LIN {X 0,Y 446.51,Z 528.86,A -85,B 0,C 180,E1 -8628.193,E2 -8628.193} C_VEL
LIN {X 0,Y 446.592,Z 528.855,A -85,B 0,C 180,E1 -8631.858,E2 -8631.858} C_VEL
LIN {X 0,Y 446.639,Z 528.845,A -85,B 0,C 180,E1 -8634.582,E2 -8634.582} C_VEL
LIN {X 0,Y 446.702,Z 528.834,A -85,B 0,C 180,E1 -8637.295,E2 -8637.295} C_VEL
LIN {X 0,Y 446.787,Z 528.83,A -85,B 0,C 180,E1 -8640,E2 -8640} C_VEL
LIN {X 0,Y 446.703,Z 528.834,A -85,B 0,C 180,E1 -8642.705,E2 -8642.705} C_VEL
LIN {X 0,Y 446.639,Z 528.846,A -85,B 0,C 180,E1 -8646.324,E2 -8646.324} C_VEL
LIN {X 0,Y 446.531,Z 528.859,A -85,B 0,C 180,E1 -8649.055,E2 -8649.055} C_VEL
LIN {X 0,Y 446.526,Z 528.859,A -85,B 0,C 180,E1 -8652.73,E2 -8652.73} C_VEL
LIN {X 0,Y 446.482,Z 528.86,A -85,B 0,C 180,E1 -8656.459,E2 -8656.459} C_VEL
LIN {X 0,Y 446.462,Z 528.872,A -85,B 0,C 180,E1 -8659.304,E2 -8659.304} C_VEL
LIN {X 0,Y 446.411,Z 528.873,A -85,B 0,C 180,E1 -8662.2,E2 -8662.2} C_VEL
LIN {X 0,Y 446.452,Z 528.872,A -85,B 0,C 180,E1 -8665.153,E2 -8665.153} C_VEL
LIN {X 0,Y 446.478,Z 528.868,A -85,B 0,C 180,E1 -8668.179,E2 -8668.179} C_VEL
LIN {X 0,Y 446.428,Z 528.877,A -85,B 0,C 180,E1 -8671.779,E2 -8671.779} C_VEL
LIN {X 0,Y 446.425,Z 528.871,A -85,B 0,C 180,E1 -8675.054,E2 -8675.054} C_VEL
LIN {X 0,Y 446.425,Z 528.874,A -85,B 0,C 180,E1 -8678.083,E2 -8678.083} C_VEL
LIN {X 0,Y 446.422,Z 528.873,A -85,B 0,C 180,E1 -8680.918,E2 -8680.918} C_VEL
LIN {X 0,Y 446.412,Z 528.878,A -85,B 0,C 180,E1 -8683.845,E2 -8683.845} C_VEL
LIN {X 0,Y 446.442,Z 528.867,A -85,B 0,C 180,E1 -8686.398,E2 -8686.398} C_VEL
LIN {X 0,Y 446.465,Z 528.87,A -85,B 0,C 180,E1 -8689.806,E2 -8689.806} C_VEL
LIN {X 0,Y 446.429,Z 528.859,A -85,B 0,C 180,E1 -8692.125,E2 -8692.125} C_VEL
LIN {X 0,Y 446.428,Z 528.877,A -85,B 0,C 180,E1 -8695.478,E2 -8695.478} C_VEL
LIN {X 0,Y 446.414,Z 528.831,A -85,B 0,C 180,E1 -8698.701,E2 -8698.701} C_VEL
LIN {X 0,Y 446.483,Z 528.871,A -85,B 0,C 180,E1 -8701.822,E2 -8701.822} C_VEL
LIN {X 0,Y 446.527,Z 529.058,A -85,B 0,C 180,E1 -8703.557,E2 -8703.557} C_VEL
LIN {X 0,Y 448.792,Z 540.632,A -85,B 0,C 180,E1 -8705.975,E2 -8705.975} C_VEL
LIN {X 0,Y 449.081,Z 544.438,A -85,B 0,C 180,E1 -8706.725,E2 -8706.725} C_VEL
LIN {X 0,Y 448.095,Z 560.858,A -85,B 0,C 180,E1 -8709.816,E2 -8709.816} C_VEL
LIN {X 0,Y 447.517,Z 573.5,A -85,B 0,C 180,E1 -8712.138,E2 -8712.138} C_VEL
LIN {X 0,Y 450.897,Z 595.443,A -85,B 0,C 180,E1 -8712.662,E2 -8712.662} C_VEL
LIN {X 0,Y 450.108,Z 681.533,A -85,B 0,C 180,E1 -8714.056,E2 -8714.056} C_VEL
LIN {X 0,Y 449.652,Z 694.781,A -85,B 0,C 180,E1 -8714.447,E2 -8714.447} C_VEL
LIN {X 0,Y 449.113,Z 708.062,A -85,B 0,C 180,E1 -8715.037,E2 -8715.037} C_VEL
LIN {X 0,Y 448.566,Z 719.218,A -85,B 0,C 180,E1 -8715.715,E2 -8715.715} C_VEL
LIN {X 0,Y 447.922,Z 730.654,A -85,B 0,C 180,E1 -8716.605,E2 -8716.605} C_VEL
LIN {X 0,Y 447.407,Z 741.258,A -85,B 0,C 180,E1 -8717.643,E2 -8717.643} C_VEL
LIN {X 0,Y 446.849,Z 749.797,A -85,B 0,C 180,E1 -8718.663,E2 -8718.663} C_VEL
LIN {X 0,Y 446.393,Z 757.677,A -85,B 0,C 180,E1 -8719.799,E2 -8719.799} C_VEL
LIN {X 0,Y 445.992,Z 765.376,A -85,B 0,C 180,E1 -8721.163,E2 -8721.163} C_VEL
LIN {X 0,Y 445.668,Z 772.472,A -85,B 0,C 180,E1 -8722.753,E2 -8722.753} C_VEL
LIN {X 0,Y 445.494,Z 776.598,A -85,B 0,C 180,E1 -8723.926,E2 -8723.926} C_VEL
LIN {X 0,Y 445.417,Z 780.807,A -85,B 0,C 180,E1 -8725.476,E2 -8725.476} C_VEL
LIN {X 0,Y 445.381,Z 782.669,A -85,B 0,C 180,E1 -8726.382,E2 -8726.382} C_VEL
LIN {X 0,Y 445.433,Z 784.067,A -85,B 0,C 180,E1 -8727.288,E2 -8727.288} C_VEL
LIN {X 0,Y 445.338,Z 785.666,A -85,B 0,C 180,E1 -8729.097,E2 -8729.097} C_VEL
LIN {X 0,Y 445.342,Z 785.882,A -85,B 0,C 180,E1 -8730.001,E2 -8730.001} C_VEL
LIN {X 0,Y 445.338,Z 785.664,A -85,B 0,C 180,E1 -8730.905,E2 -8730.905} C_VEL
LIN {X 0,Y 445.433,Z 784.061,A -85,B 0,C 180,E1 -8732.714,E2 -8732.714} C_VEL
LIN {X 0,Y 445.381,Z 782.661,A -85,B 0,C 180,E1 -8733.62,E2 -8733.62} C_VEL
LIN {X 0,Y 445.482,Z 779.728,A -85,B 0,C 180,E1 -8734.978,E2 -8734.978} C_VEL
LIN {X 0,Y 445.576,Z 774.321,A -85,B 0,C 180,E1 -8736.749,E2 -8736.749} C_VEL
LIN {X 0,Y 445.848,Z 768.627,A -85,B 0,C 180,E1 -8738.157,E2 -8738.157} C_VEL
LIN {X 0,Y 446.16,Z 761.723,A -85,B 0,C 180,E1 -8739.521,E2 -8739.521} C_VEL
LIN {X 0,Y 446.611,Z 753.086,A -85,B 0,C 180,E1 -8740.886,E2 -8740.886} C_VEL
LIN {X 0,Y 447.213,Z 744.234,A -85,B 0,C 180,E1 -8742.019,E2 -8742.019} C_VEL
LIN {X 0,Y 447.682,Z 735.241,A -85,B 0,C 180,E1 -8742.972,E2 -8742.972} C_VEL
LIN {X 0,Y 448.293,Z 723.88,A -85,B 0,C 180,E1 -8743.948,E2 -8743.948} C_VEL
LIN {X 0,Y 448.894,Z 712.012,A -85,B 0,C 180,E1 -8744.74,E2 -8744.74} C_VEL
LIN {X 0,Y 449.493,Z 699.667,A -85,B 0,C 180,E1 -8745.357,E2 -8745.357} C_VEL
LIN {X 0,Y 449.947,Z 686.981,A -85,B 0,C 180,E1 -8745.806,E2 -8745.806} C_VEL
LIN {X 0,Y 450.202,Z 673.707,A -85,B 0,C 180,E1 -8746.087,E2 -8746.087} C_VEL
LIN {X 0,Y 450.721,Z 593.516,A -85,B 0,C 180,E1 -8747.374,E2 -8747.374} C_VEL
LIN {X 0,Y 447.503,Z 573.499,A -85,B 0,C 180,E1 -8747.859,E2 -8747.859} C_VEL
LIN {X 0,Y 448.186,Z 559.56,A -85,B 0,C 180,E1 -8750.421,E2 -8750.421} C_VEL
LIN {X 0,Y 449.08,Z 544.406,A -85,B 0,C 180,E1 -8753.276,E2 -8753.276} C_VEL
LIN {X 0,Y 448.611,Z 539.586,A -85,B 0,C 180,E1 -8754.233,E2 -8754.233} C_VEL
LIN {X 0,Y 446.536,Z 529.053,A -85,B 0,C 180,E1 -8756.444,E2 -8756.444} C_VEL
LIN {X 0,Y 446.452,Z 528.857,A -85,B 0,C 180,E1 -8759.21,E2 -8759.21} C_VEL
LIN {X 0,Y 446.426,Z 528.879,A -85,B 0,C 180,E1 -8762.362,E2 -8762.362} C_VEL
LIN {X 0,Y 446.423,Z 528.875,A -85,B 0,C 180,E1 -8765.626,E2 -8765.626} C_VEL
LIN {X 0,Y 446.448,Z 528.872,A -85,B 0,C 180,E1 -8769.027,E2 -8769.027} C_VEL
LIN {X 0,Y 446.438,Z 528.875,A -85,B 0,C 180,E1 -8772.278,E2 -8772.278} C_VEL
LIN {X 0,Y 446.455,Z 528.872,A -85,B 0,C 180,E1 -8775.104,E2 -8775.104} C_VEL
LIN {X 0,Y 446.431,Z 528.876,A -85,B 0,C 180,E1 -8778.609,E2 -8778.609} C_VEL
LIN {X 0,Y 446.464,Z 528.87,A -85,B 0,C 180,E1 -8780.975,E2 -8780.975} C_VEL
LIN {X 0,Y 446.424,Z 528.88,A -85,B 0,C 180,E1 -8784.374,E2 -8784.374} C_VEL
LIN {X 0,Y 446.426,Z 528.877,A -85,B 0,C 180,E1 -8787.639,E2 -8787.639} C_VEL
LIN {X 0,Y 446.453,Z 528.876,A -85,B 0,C 180,E1 -8790.791,E2 -8790.791} C_VEL
LIN {X 0,Y 446.536,Z 529.061,A -85,B 0,C 180,E1 -8792.271,E2 -8792.271} C_VEL
LIN {X 0,Y 448.78,Z 539.14,A -85,B 0,C 180,E1 -8793.993,E2 -8793.993} C_VEL
LIN {X 0,Y 449.498,Z 544.011,A -85,B 0,C 180,E1 -8794.782,E2 -8794.782} C_VEL
LIN {X 0,Y 448.867,Z 564.635,A -85,B 0,C 180,E1 -8797.928,E2 -8797.928} C_VEL
LIN {X 0,Y 448.11,Z 586.321,A -85,B 0,C 180,E1 -8801.245,E2 -8801.245} C_VEL
LIN {X 0,Y 447.44,Z 609.001,A -85,B 0,C 180,E1 -8804.746,E2 -8804.746} C_VEL
LIN {X 0,Y 447.231,Z 616.994,A -85,B 0,C 180,E1 -8805.934,E2 -8805.934} C_VEL
LIN {X 0,Y 448.935,Z 631.407,A -85,B 0,C 180,E1 -8806.294,E2 -8806.294} C_VEL
LIN {X 0,Y 448.157,Z 697.089,A -85,B 0,C 180,E1 -8807.548,E2 -8807.548} C_VEL
LIN {X 0,Y 447.884,Z 707.461,A -85,B 0,C 180,E1 -8807.885,E2 -8807.885} C_VEL
LIN {X 0,Y 447.61,Z 717.158,A -85,B 0,C 180,E1 -8808.337,E2 -8808.337} C_VEL
LIN {X 0,Y 447.278,Z 728.032,A -85,B 0,C 180,E1 -8809.017,E2 -8809.017} C_VEL
LIN {X 0,Y 446.889,Z 737.516,A -85,B 0,C 180,E1 -8809.809,E2 -8809.809} C_VEL
LIN {X 0,Y 446.624,Z 744.205,A -85,B 0,C 180,E1 -8810.49,E2 -8810.49} C_VEL
LIN {X 0,Y 446.26,Z 751.577,A -85,B 0,C 180,E1 -8811.396,E2 -8811.396} C_VEL
LIN {X 0,Y 445.99,Z 757.653,A -85,B 0,C 180,E1 -8812.302,E2 -8812.302} C_VEL
LIN {X 0,Y 445.825,Z 763.632,A -85,B 0,C 180,E1 -8813.393,E2 -8813.393} C_VEL
LIN {X 0,Y 445.656,Z 768.771,A -85,B 0,C 180,E1 -8814.571,E2 -8814.571} C_VEL
LIN {X 0,Y 445.485,Z 773.124,A -85,B 0,C 180,E1 -8815.929,E2 -8815.929} C_VEL
LIN {X 0,Y 445.449,Z 776.133,A -85,B 0,C 180,E1 -8817.287,E2 -8817.287} C_VEL
LIN {X 0,Y 445.356,Z 777.465,A -85,B 0,C 180,E1 -8818.191,E2 -8818.191} C_VEL
LIN {X 0,Y 445.314,Z 778.286,A -85,B 0,C 180,E1 -8819.096,E2 -8819.096} C_VEL
LIN {X 0,Y 445.315,Z 778.581,A -85,B 0,C 180,E1 -8820,E2 -8820} C_VEL
LIN {X 0,Y 445.315,Z 778.281,A -85,B 0,C 180,E1 -8820.904,E2 -8820.904} C_VEL
LIN {X 0,Y 445.357,Z 777.461,A -85,B 0,C 180,E1 -8821.809,E2 -8821.809} C_VEL
LIN {X 0,Y 445.449,Z 776.132,A -85,B 0,C 180,E1 -8822.713,E2 -8822.713} C_VEL
LIN {X 0,Y 445.465,Z 773.118,A -85,B 0,C 180,E1 -8824.071,E2 -8824.071} C_VEL
LIN {X 0,Y 445.625,Z 768.766,A -85,B 0,C 180,E1 -8825.43,E2 -8825.43} C_VEL
LIN {X 0,Y 445.781,Z 763.037,A -85,B 0,C 180,E1 -8826.725,E2 -8826.725} C_VEL
LIN {X 0,Y 445.94,Z 757.662,A -85,B 0,C 180,E1 -8827.699,E2 -8827.699} C_VEL
LIN {X 0,Y 446.211,Z 751.59,A -85,B 0,C 180,E1 -8828.605,E2 -8828.605} C_VEL
LIN {X 0,Y 446.515,Z 744.23,A -85,B 0,C 180,E1 -8829.513,E2 -8829.513} C_VEL
LIN {X 0,Y 446.924,Z 735.167,A -85,B 0,C 180,E1 -8830.419,E2 -8830.419} C_VEL
LIN {X 0,Y 447.32,Z 724.744,A -85,B 0,C 180,E1 -8831.211,E2 -8831.211} C_VEL
LIN {X 0,Y 447.566,Z 716.17,A -85,B 0,C 180,E1 -8831.722,E2 -8831.722} C_VEL
LIN {X 0,Y 447.778,Z 706.821,A -85,B 0,C 180,E1 -8832.147,E2 -8832.147} C_VEL
LIN {X 0,Y 448.033,Z 696.114,A -85,B 0,C 180,E1 -8832.485,E2 -8832.485} C_VEL
LIN {X 0,Y 448.615,Z 629.959,A -85,B 0,C 180,E1 -8833.69,E2 -8833.69} C_VEL
LIN {X 0,Y 447.022,Z 616.645,A -85,B 0,C 180,E1 -8834.006,E2 -8834.006} C_VEL
LIN {X 0,Y 447.552,Z 598.063,A -85,B 0,C 180,E1 -8836.901,E2 -8836.901} C_VEL
LIN {X 0,Y 448.343,Z 577.229,A -85,B 0,C 180,E1 -8840.173,E2 -8840.173} C_VEL
LIN {X 0,Y 449.038,Z 557.569,A -85,B 0,C 180,E1 -8843.278,E2 -8843.278} C_VEL
LIN {X 0,Y 449.527,Z 545.318,A -85,B 0,C 180,E1 -8845.216,E2 -8845.216} C_VEL
LIN {X 0,Y 448.529,Z 538.743,A -85,B 0,C 180,E1 -8846.316,E2 -8846.316} C_VEL
LIN {X 0,Y 446.533,Z 528.964,A -85,B 0,C 180,E1 -8848.027,E2 -8848.027} C_VEL
LIN {X 0,Y 446.42,Z 528.879,A -85,B 0,C 180,E1 -8851.3,E2 -8851.3} C_VEL
LIN {X 0,Y 446.433,Z 528.873,A -85,B 0,C 180,E1 -8854.523,E2 -8854.523} C_VEL
LIN {X 0,Y 446.434,Z 528.872,A -85,B 0,C 180,E1 -8858.082,E2 -8858.082} C_VEL
LIN {X 0,Y 446.427,Z 528.861,A -85,B 0,C 180,E1 -8860.917,E2 -8860.917} C_VEL
LIN {X 0,Y 446.403,Z 528.866,A -85,B 0,C 180,E1 -8863.846,E2 -8863.846} C_VEL
LIN {X 0,Y 446.402,Z 528.876,A -85,B 0,C 180,E1 -8866.403,E2 -8866.403} C_VEL
LIN {X 0,Y 446.431,Z 528.864,A -85,B 0,C 180,E1 -8869.082,E2 -8869.082} C_VEL
LIN {X 0,Y 446.411,Z 528.872,A -85,B 0,C 180,E1 -8872.121,E2 -8872.121} C_VEL
LIN {X 0,Y 446.427,Z 528.871,A -85,B 0,C 180,E1 -8875.476,E2 -8875.476} C_VEL
LIN {X 0,Y 446.42,Z 528.875,A -85,B 0,C 180,E1 -8878.699,E2 -8878.699} C_VEL
LIN {X 0,Y 446.489,Z 528.867,A -85,B 0,C 180,E1 -8881.821,E2 -8881.821} C_VEL
LIN {X 0,Y 446.454,Z 528.871,A -85,B 0,C 180,E1 -8884.847,E2 -8884.847} C_VEL
LIN {X 0,Y 446.478,Z 529.008,A -85,B 0,C 180,E1 -8887.437,E2 -8887.437} C_VEL
LIN {X 0,Y 448.136,Z 537.779,A -85,B 0,C 180,E1 -8889.577,E2 -8889.577} C_VEL
LIN {X 0,Y 448.116,Z 539.979,A -85,B 0,C 180,E1 -8890.073,E2 -8890.073} C_VEL
LIN {X 0,Y 447.429,Z 543.234,A -85,B 0,C 180,E1 -8890.675,E2 -8890.675} C_VEL
LIN {X 0,Y 445.584,Z 548.544,A -85,B 0,C 180,E1 -8891.354,E2 -8891.354} C_VEL
LIN {X 0,Y 443.803,Z 554.744,A -85,B 0,C 180,E1 -8891.883,E2 -8891.883} C_VEL
LIN {X 0,Y 443.187,Z 559.936,A -85,B 0,C 180,E1 -8892.167,E2 -8892.167} C_VEL
LIN {X 0,Y 443.431,Z 563.572,A -85,B 0,C 180,E1 -8892.287,E2 -8892.287} C_VEL
LIN {X 0,Y 444.253,Z 568.245,A -85,B 0,C 180,E1 -8892.399,E2 -8892.399} C_VEL
LIN {X 0,Y 443.384,Z 657.163,A -85,B 0,C 180,E1 -8893.865,E2 -8893.865} C_VEL
LIN {X 0,Y 442.99,Z 671.026,A -85,B 0,C 180,E1 -8894.294,E2 -8894.294} C_VEL
LIN {X 0,Y 442.503,Z 683.424,A -85,B 0,C 180,E1 -8894.866,E2 -8894.866} C_VEL
LIN {X 0,Y 441.942,Z 695.269,A -85,B 0,C 180,E1 -8895.612,E2 -8895.612} C_VEL
LIN {X 0,Y 441.388,Z 706.671,A -85,B 0,C 180,E1 -8896.537,E2 -8896.537} C_VEL
LIN {X 0,Y 440.768,Z 716.867,A -85,B 0,C 180,E1 -8897.569,E2 -8897.569} C_VEL
LIN {X 0,Y 440.149,Z 726.052,A -85,B 0,C 180,E1 -8898.72,E2 -8898.72} C_VEL
LIN {X 0,Y 439.552,Z 734.97,A -85,B 0,C 180,E1 -8900.102,E2 -8900.102} C_VEL
LIN {X 0,Y 439.104,Z 742.146,A -85,B 0,C 180,E1 -8901.485,E2 -8901.485} C_VEL
LIN {X 0,Y 438.788,Z 746.99,A -85,B 0,C 180,E1 -8902.637,E2 -8902.637} C_VEL
LIN {X 0,Y 438.686,Z 751.69,A -85,B 0,C 180,E1 -8904.022,E2 -8904.022} C_VEL
LIN {X 0,Y 438.424,Z 755.291,A -85,B 0,C 180,E1 -8905.402,E2 -8905.402} C_VEL
LIN {X 0,Y 438.428,Z 757.148,A -85,B 0,C 180,E1 -8906.323,E2 -8906.323} C_VEL
LIN {X 0,Y 438.395,Z 758.551,A -85,B 0,C 180,E1 -8907.243,E2 -8907.243} C_VEL
LIN {X 0,Y 438.255,Z 760.167,A -85,B 0,C 180,E1 -8909.08,E2 -8909.08} C_VEL
LIN {X 0,Y 438.254,Z 760.402,A -85,B 0,C 180,E1 -8909.999,E2 -8909.999} C_VEL
LIN {X 0,Y 438.255,Z 760.216,A -85,B 0,C 180,E1 -8910.918,E2 -8910.918} C_VEL
LIN {X 0,Y 438.392,Z 758.667,A -85,B 0,C 180,E1 -8912.756,E2 -8912.756} C_VEL
LIN {X 0,Y 438.413,Z 757.314,A -85,B 0,C 180,E1 -8913.676,E2 -8913.676} C_VEL
LIN {X 0,Y 438.481,Z 754.45,A -85,B 0,C 180,E1 -8915.057,E2 -8915.057} C_VEL
LIN {X 0,Y 438.693,Z 750.563,A -85,B 0,C 180,E1 -8916.438,E2 -8916.438} C_VEL
LIN {X 0,Y 438.902,Z 745.555,A -85,B 0,C 180,E1 -8917.822,E2 -8917.822} C_VEL
LIN {X 0,Y 439.321,Z 739.248,A -85,B 0,C 180,E1 -8919.205,E2 -8919.205} C_VEL
LIN {X 0,Y 439.803,Z 731.349,A -85,B 0,C 180,E1 -8920.588,E2 -8920.588} C_VEL
LIN {X 0,Y 440.285,Z 723.299,A -85,B 0,C 180,E1 -8921.742,E2 -8921.742} C_VEL
LIN {X 0,Y 441.015,Z 713.467,A -85,B 0,C 180,E1 -8922.89,E2 -8922.89} C_VEL
LIN {X 0,Y 441.542,Z 702.694,A -85,B 0,C 180,E1 -8923.907,E2 -8923.907} C_VEL
LIN {X 0,Y 442.135,Z 691.584,A -85,B 0,C 180,E1 -8924.733,E2 -8924.733} C_VEL
LIN {X 0,Y 442.709,Z 679.604,A -85,B 0,C 180,E1 -8925.42,E2 -8925.42} C_VEL
LIN {X 0,Y 443.122,Z 666.471,A -85,B 0,C 180,E1 -8925.966,E2 -8925.966} C_VEL
LIN {X 0,Y 443.533,Z 653.261,A -85,B 0,C 180,E1 -8926.305,E2 -8926.305} C_VEL
LIN {X 0,Y 444.113,Z 567.022,A -85,B 0,C 180,E1 -8927.721,E2 -8927.721} C_VEL
LIN {X 0,Y 440.768,Z 550.156,A -85,B 0,C 180,E1 -8928.171,E2 -8928.171} C_VEL
LIN {X 0,Y 440.78,Z 547.921,A -85,B 0,C 180,E1 -8928.595,E2 -8928.595} C_VEL
LIN {X 0,Y 441.2,Z 539.437,A -85,B 0,C 180,E1 -8930.513,E2 -8930.513} C_VEL
LIN {X 0,Y 439.437,Z 529.822,A -85,B 0,C 180,E1 -8932.912,E2 -8932.912} C_VEL
LIN {X 0,Y 439.433,Z 529.742,A -85,B 0,C 180,E1 -8936.41,E2 -8936.41} C_VEL
LIN {X 0,Y 439.417,Z 529.744,A -85,B 0,C 180,E1 -8938.672,E2 -8938.672} C_VEL
LIN {X 0,Y 439.369,Z 529.753,A -85,B 0,C 180,E1 -8942.03,E2 -8942.03} C_VEL
LIN {X 0,Y 439.394,Z 529.752,A -85,B 0,C 180,E1 -8945.34,E2 -8945.34} C_VEL
LIN {X 0,Y 439.387,Z 529.75,A -85,B 0,C 180,E1 -8948.593,E2 -8948.593} C_VEL
LIN {X 0,Y 439.386,Z 529.751,A -85,B 0,C 180,E1 -8951.256,E2 -8951.256} C_VEL
LIN {X 0,Y 439.401,Z 529.741,A -85,B 0,C 180,E1 -8954.728,E2 -8954.728} C_VEL
LIN {X 0,Y 439.393,Z 529.752,A -85,B 0,C 180,E1 -8957.795,E2 -8957.795} C_VEL
LIN {X 0,Y 439.447,Z 529.734,A -85,B 0,C 180,E1 -8960.229,E2 -8960.229} C_VEL
LIN {X 0,Y 439.373,Z 529.756,A -85,B 0,C 180,E1 -8963.712,E2 -8963.712} C_VEL
LIN {X 0,Y 439.367,Z 529.754,A -85,B 0,C 180,E1 -8967.053,E2 -8967.053} C_VEL
LIN {X 0,Y 439.39,Z 529.749,A -85,B 0,C 180,E1 -8970.275,E2 -8970.275} C_VEL
LIN {X 0,Y 439.427,Z 529.748,A -85,B 0,C 180,E1 -8973.588,E2 -8973.588} C_VEL
LIN {X 0,Y 439.38,Z 529.748,A -85,B 0,C 180,E1 -8976.429,E2 -8976.429} C_VEL
LIN {X 0,Y 439.382,Z 529.752,A -85,B 0,C 180,E1 -8979.397,E2 -8979.397} C_VEL
LIN {X 0,Y 439.424,Z 529.741,A -85,B 0,C 180,E1 -8982.309,E2 -8982.309} C_VEL
LIN {X 0,Y 439.44,Z 529.741,A -85,B 0,C 180,E1 -8985.174,E2 -8985.174} C_VEL
LIN {X 0,Y 439.476,Z 529.738,A -85,B 0,C 180,E1 -8988.001,E2 -8988.001} C_VEL
LIN {X 0,Y 439.54,Z 529.734,A -85,B 0,C 180,E1 -8991.726,E2 -8991.726} C_VEL
LIN {X 0,Y 439.614,Z 529.72,A -85,B 0,C 180,E1 -8994.496,E2 -8994.496} C_VEL
LIN {X 0,Y 439.628,Z 529.718,A -85,B 0,C 180,E1 -8998.168,E2 -8998.168} C_VEL
LIN {X 0,Y 439.757,Z 529.706,A -85,B 0,C 180,E1 -9000,E2 -9000} C_VEL
LIN {X 0,Y 439.649,Z 529.712,A -85,B 0,C 180,E1 -9002.749,E2 -9002.749} C_VEL
LIN {X 0,Y 439.61,Z 529.721,A -85,B 0,C 180,E1 -9006.425,E2 -9006.425} C_VEL
LIN {X 0,Y 439.493,Z 529.737,A -85,B 0,C 180,E1 -9009.202,E2 -9009.202} C_VEL
LIN {X 0,Y 439.496,Z 529.735,A -85,B 0,C 180,E1 -9012.727,E2 -9012.727} C_VEL
LIN {X 0,Y 439.44,Z 529.737,A -85,B 0,C 180,E1 -9016.349,E2 -9016.349} C_VEL
LIN {X 0,Y 439.424,Z 529.751,A -85,B 0,C 180,E1 -9019.625,E2 -9019.625} C_VEL
LIN {X 0,Y 439.358,Z 529.75,A -85,B 0,C 180,E1 -9022.576,E2 -9022.576} C_VEL
LIN {X 0,Y 439.399,Z 529.752,A -85,B 0,C 180,E1 -9025.585,E2 -9025.585} C_VEL
LIN {X 0,Y 439.411,Z 529.747,A -85,B 0,C 180,E1 -9028.674,E2 -9028.674} C_VEL
LIN {X 0,Y 439.375,Z 529.754,A -85,B 0,C 180,E1 -9032.034,E2 -9032.034} C_VEL
LIN {X 0,Y 439.39,Z 529.748,A -85,B 0,C 180,E1 -9035.342,E2 -9035.342} C_VEL
LIN {X 0,Y 439.385,Z 529.749,A -85,B 0,C 180,E1 -9038.595,E2 -9038.595} C_VEL
LIN {X 0,Y 439.383,Z 529.752,A -85,B 0,C 180,E1 -9041.258,E2 -9041.258} C_VEL
LIN {X 0,Y 439.4,Z 529.748,A -85,B 0,C 180,E1 -9044.73,E2 -9044.73} C_VEL
LIN {X 0,Y 439.409,Z 529.749,A -85,B 0,C 180,E1 -9047.799,E2 -9047.799} C_VEL
LIN {X 0,Y 439.447,Z 529.739,A -85,B 0,C 180,E1 -9050.231,E2 -9050.231} C_VEL
LIN {X 0,Y 439.374,Z 529.748,A -85,B 0,C 180,E1 -9053.714,E2 -9053.714} C_VEL
LIN {X 0,Y 439.37,Z 529.733,A -85,B 0,C 180,E1 -9057.055,E2 -9057.055} C_VEL
LIN {X 0,Y 439.38,Z 529.723,A -85,B 0,C 180,E1 -9060.275,E2 -9060.275} C_VEL
LIN {X 0,Y 439.47,Z 529.836,A -85,B 0,C 180,E1 -9063.272,E2 -9063.272} C_VEL
LIN {X 0,Y 441.813,Z 541.718,A -85,B 0,C 180,E1 -9065.821,E2 -9065.821} C_VEL
LIN {X 0,Y 442.142,Z 545.523,A -85,B 0,C 180,E1 -9066.586,E2 -9066.586} C_VEL
LIN {X 0,Y 441.101,Z 562.606,A -85,B 0,C 180,E1 -9069.856,E2 -9069.856} C_VEL
LIN {X 0,Y 440.59,Z 573.219,A -85,B 0,C 180,E1 -9071.841,E2 -9071.841} C_VEL
LIN {X 0,Y 442.189,Z 582.977,A -85,B 0,C 180,E1 -9072.105,E2 -9072.105} C_VEL
LIN {X 0,Y 444.109,Z 596.39,A -85,B 0,C 180,E1 -9072.407,E2 -9072.407} C_VEL
LIN {X 0,Y 443.298,Z 681.339,A -85,B 0,C 180,E1 -9073.805,E2 -9073.805} C_VEL
LIN {X 0,Y 442.821,Z 694.584,A -85,B 0,C 180,E1 -9074.201,E2 -9074.201} C_VEL
LIN {X 0,Y 442.312,Z 706.741,A -85,B 0,C 180,E1 -9074.743,E2 -9074.743} C_VEL
LIN {X 0,Y 441.681,Z 719.017,A -85,B 0,C 180,E1 -9075.487,E2 -9075.487} C_VEL
LIN {X 0,Y 441.048,Z 729.687,A -85,B 0,C 180,E1 -9076.323,E2 -9076.323} C_VEL
LIN {X 0,Y 440.443,Z 741.055,A -85,B 0,C 180,E1 -9077.444,E2 -9077.444} C_VEL
LIN {X 0,Y 439.873,Z 749.594,A -85,B 0,C 180,E1 -9078.48,E2 -9078.48} C_VEL
LIN {X 0,Y 439.371,Z 757.473,A -85,B 0,C 180,E1 -9079.634,E2 -9079.634} C_VEL
LIN {X 0,Y 438.937,Z 765.171,A -85,B 0,C 180,E1 -9081.02,E2 -9081.02} C_VEL
LIN {X 0,Y 438.606,Z 772.267,A -85,B 0,C 180,E1 -9082.636,E2 -9082.636} C_VEL
LIN {X 0,Y 438.393,Z 776.825,A -85,B 0,C 180,E1 -9083.967,E2 -9083.967} C_VEL
LIN {X 0,Y 438.346,Z 780.603,A -85,B 0,C 180,E1 -9085.403,E2 -9085.403} C_VEL
LIN {X 0,Y 438.283,Z 782.465,A -85,B 0,C 180,E1 -9086.323,E2 -9086.323} C_VEL
LIN {X 0,Y 438.341,Z 783.862,A -85,B 0,C 180,E1 -9087.244,E2 -9087.244} C_VEL
LIN {X 0,Y 438.252,Z 785.462,A -85,B 0,C 180,E1 -9089.082,E2 -9089.082} C_VEL
LIN {X 0,Y 438.253,Z 785.678,A -85,B 0,C 180,E1 -9090.001,E2 -9090.001} C_VEL
LIN {X 0,Y 438.278,Z 784.851,A -85,B 0,C 180,E1 -9091.839,E2 -9091.839} C_VEL
LIN {X 0,Y 438.341,Z 783.856,A -85,B 0,C 180,E1 -9092.758,E2 -9092.758} C_VEL
LIN {X 0,Y 438.283,Z 782.456,A -85,B 0,C 180,E1 -9093.678,E2 -9093.678} C_VEL
LIN {X 0,Y 438.392,Z 779.522,A -85,B 0,C 180,E1 -9095.059,E2 -9095.059} C_VEL
LIN {X 0,Y 438.449,Z 775.547,A -85,B 0,C 180,E1 -9096.443,E2 -9096.443} C_VEL
LIN {X 0,Y 438.724,Z 769.433,A -85,B 0,C 180,E1 -9098.058,E2 -9098.058} C_VEL
LIN {X 0,Y 439.066,Z 762.753,A -85,B 0,C 180,E1 -9099.444,E2 -9099.444} C_VEL
LIN {X 0,Y 439.523,Z 754.467,A -85,B 0,C 180,E1 -9100.83,E2 -9100.83} C_VEL
LIN {X 0,Y 440.111,Z 745.977,A -85,B 0,C 180,E1 -9101.982,E2 -9101.982} C_VEL
LIN {X 0,Y 440.68,Z 735.869,A -85,B 0,C 180,E1 -9103.098,E2 -9103.098} C_VEL
LIN {X 0,Y 441.295,Z 725.101,A -85,B 0,C 180,E1 -9104.057,E2 -9104.057} C_VEL
LIN {X 0,Y 441.922,Z 713.728,A -85,B 0,C 180,E1 -9104.86,E2 -9104.86} C_VEL
LIN {X 0,Y 442.536,Z 702.061,A -85,B 0,C 180,E1 -9105.487,E2 -9105.487} C_VEL
LIN {X 0,Y 443.031,Z 688.601,A -85,B 0,C 180,E1 -9106,E2 -9106} C_VEL
LIN {X 0,Y 443.398,Z 675.272,A -85,B 0,C 180,E1 -9106.311,E2 -9106.311} C_VEL
LIN {X 0,Y 443.994,Z 594.706,A -85,B 0,C 180,E1 -9107.622,E2 -9107.622} C_VEL
LIN {X 0,Y 440.562,Z 573.531,A -85,B 0,C 180,E1 -9108.133,E2 -9108.133} C_VEL
LIN {X 0,Y 440.689,Z 570.679,A -85,B 0,C 180,E1 -9108.6,E2 -9108.6} C_VEL
LIN {X 0,Y 441.86,Z 550.549,A -85,B 0,C 180,E1 -9112.442,E2 -9112.442} C_VEL
LIN {X 0,Y 442.137,Z 544.223,A -85,B 0,C 180,E1 -9113.664,E2 -9113.664} C_VEL
LIN {X 0,Y 440.358,Z 534.063,A -85,B 0,C 180,E1 -9115.776,E2 -9115.776} C_VEL
LIN {X 0,Y 439.482,Z 529.843,A -85,B 0,C 180,E1 -9116.729,E2 -9116.729} C_VEL
LIN {X 0,Y 439.386,Z 529.741,A -85,B 0,C 180,E1 -9119.726,E2 -9119.726} C_VEL
LIN {X 0,Y 439.376,Z 529.753,A -85,B 0,C 180,E1 -9122.946,E2 -9122.946} C_VEL
LIN {X 0,Y 439.377,Z 529.756,A -85,B 0,C 180,E1 -9126.287,E2 -9126.287} C_VEL
LIN {X 0,Y 439.405,Z 529.752,A -85,B 0,C 180,E1 -9129.849,E2 -9129.849} C_VEL
LIN {X 0,Y 439.385,Z 529.754,A -85,B 0,C 180,E1 -9132.627,E2 -9132.627} C_VEL
LIN {X 0,Y 439.403,Z 529.75,A -85,B 0,C 180,E1 -9135.271,E2 -9135.271} C_VEL
LIN {X 0,Y 439.392,Z 529.752,A -85,B 0,C 180,E1 -9138.743,E2 -9138.743} C_VEL
LIN {X 0,Y 439.389,Z 529.753,A -85,B 0,C 180,E1 -9141.606,E2 -9141.606} C_VEL
LIN {X 0,Y 439.404,Z 529.751,A -85,B 0,C 180,E1 -9144.844,E2 -9144.844} C_VEL
LIN {X 0,Y 439.376,Z 529.757,A -85,B 0,C 180,E1 -9148.14,E2 -9148.14} C_VEL
LIN {X 0,Y 439.458,Z 529.785,A -85,B 0,C 180,E1 -9151.792,E2 -9151.792} C_VEL
LIN {X 0,Y 439.61,Z 530.432,A -85,B 0,C 180,E1 -9152.024,E2 -9152.024} C_VEL
LIN {X 0,Y 441.68,Z 539.177,A -85,B 0,C 180,E1 -9153.542,E2 -9153.542} C_VEL
LIN {X 0,Y 442.705,Z 545.655,A -85,B 0,C 180,E1 -9154.619,E2 -9154.619} C_VEL
LIN {X 0,Y 442.015,Z 566.31,A -85,B 0,C 180,E1 -9157.813,E2 -9157.813} C_VEL
LIN {X 0,Y 441.186,Z 588.036,A -85,B 0,C 180,E1 -9161.181,E2 -9161.181} C_VEL
LIN {X 0,Y 440.478,Z 610.836,A -85,B 0,C 180,E1 -9164.736,E2 -9164.736} C_VEL
LIN {X 0,Y 440.288,Z 616.892,A -85,B 0,C 180,E1 -9165.646,E2 -9165.646} C_VEL
LIN {X 0,Y 442.102,Z 631.443,A -85,B 0,C 180,E1 -9166.043,E2 -9166.043} C_VEL
LIN {X 0,Y 441.214,Z 697.846,A -85,B 0,C 180,E1 -9167.348,E2 -9167.348} C_VEL
LIN {X 0,Y 440.964,Z 707.987,A -85,B 0,C 180,E1 -9167.692,E2 -9167.692} C_VEL
LIN {X 0,Y 440.668,Z 718.644,A -85,B 0,C 180,E1 -9168.209,E2 -9168.209} C_VEL
LIN {X 0,Y 440.208,Z 729.73,A -85,B 0,C 180,E1 -9168.955,E2 -9168.955} C_VEL
LIN {X 0,Y 439.913,Z 737.717,A -85,B 0,C 180,E1 -9169.646,E2 -9169.646} C_VEL
LIN {X 0,Y 439.625,Z 744.369,A -85,B 0,C 180,E1 -9170.337,E2 -9170.337} C_VEL
LIN {X 0,Y 439.236,Z 751.71,A -85,B 0,C 180,E1 -9171.257,E2 -9171.257} C_VEL
LIN {X 0,Y 438.94,Z 757.766,A -85,B 0,C 180,E1 -9172.178,E2 -9172.178} C_VEL
LIN {X 0,Y 438.769,Z 763.612,A -85,B 0,C 180,E1 -9173.262,E2 -9173.262} C_VEL
LIN {X 0,Y 438.602,Z 768.872,A -85,B 0,C 180,E1 -9174.483,E2 -9174.483} C_VEL
LIN {X 0,Y 438.389,Z 773.216,A -85,B 0,C 180,E1 -9175.863,E2 -9175.863} C_VEL
LIN {X 0,Y 438.379,Z 776.224,A -85,B 0,C 180,E1 -9177.243,E2 -9177.243} C_VEL
LIN {X 0,Y 438.279,Z 777.542,A -85,B 0,C 180,E1 -9178.162,E2 -9178.162} C_VEL
LIN {X 0,Y 438.229,Z 778.351,A -85,B 0,C 180,E1 -9179.081,E2 -9179.081} C_VEL
LIN {X 0,Y 438.227,Z 778.636,A -85,B 0,C 180,E1 -9180,E2 -9180} C_VEL
LIN {X 0,Y 438.23,Z 778.326,A -85,B 0,C 180,E1 -9180.919,E2 -9180.919} C_VEL
LIN {X 0,Y 438.28,Z 777.483,A -85,B 0,C 180,E1 -9181.838,E2 -9181.838} C_VEL
LIN {X 0,Y 438.361,Z 776.13,A -85,B 0,C 180,E1 -9182.757,E2 -9182.757} C_VEL
LIN {X 0,Y 438.372,Z 773.078,A -85,B 0,C 180,E1 -9184.137,E2 -9184.137} C_VEL
LIN {X 0,Y 438.551,Z 768.665,A -85,B 0,C 180,E1 -9185.518,E2 -9185.518} C_VEL
LIN {X 0,Y 438.707,Z 763.306,A -85,B 0,C 180,E1 -9186.749,E2 -9186.749} C_VEL
LIN {X 0,Y 438.894,Z 757.451,A -85,B 0,C 180,E1 -9187.823,E2 -9187.823} C_VEL
LIN {X 0,Y 439.16,Z 751.316,A -85,B 0,C 180,E1 -9188.745,E2 -9188.745} C_VEL
LIN {X 0,Y 439.555,Z 742.888,A -85,B 0,C 180,E1 -9189.781,E2 -9189.781} C_VEL
LIN {X 0,Y 439.993,Z 733.272,A -85,B 0,C 180,E1 -9190.701,E2 -9190.701} C_VEL
LIN {X 0,Y 440.315,Z 724.079,A -85,B 0,C 180,E1 -9191.392,E2 -9191.392} C_VEL
LIN {X 0,Y 440.611,Z 714.238,A -85,B 0,C 180,E1 -9191.968,E2 -9191.968} C_VEL
LIN {X 0,Y 440.87,Z 702.638,A -85,B 0,C 180,E1 -9192.457,E2 -9192.457} C_VEL
LIN {X 0,Y 441.142,Z 689.902,A -85,B 0,C 180,E1 -9192.771,E2 -9192.771} C_VEL
LIN {X 0,Y 441.605,Z 630.077,A -85,B 0,C 180,E1 -9193.88,E2 -9193.88} C_VEL
LIN {X 0,Y 440.009,Z 616.661,A -85,B 0,C 180,E1 -9194.207,E2 -9194.207} C_VEL
LIN {X 0,Y 440.583,Z 598.143,A -85,B 0,C 180,E1 -9197.116,E2 -9197.116} C_VEL
LIN {X 0,Y 441.402,Z 576.791,A -85,B 0,C 180,E1 -9200.505,E2 -9200.505} C_VEL
LIN {X 0,Y 442.143,Z 556.985,A -85,B 0,C 180,E1 -9203.663,E2 -9203.663} C_VEL
LIN {X 0,Y 442.576,Z 546.183,A -85,B 0,C 180,E1 -9205.389,E2 -9205.389} C_VEL
LIN {X 0,Y 440.813,Z 536.225,A -85,B 0,C 180,E1 -9207.085,E2 -9207.085} C_VEL
LIN {X 0,Y 439.484,Z 529.839,A -85,B 0,C 180,E1 -9208.236,E2 -9208.236} C_VEL
LIN {X 0,Y 439.377,Z 529.757,A -85,B 0,C 180,E1 -9211.86,E2 -9211.86} C_VEL
LIN {X 0,Y 439.404,Z 529.751,A -85,B 0,C 180,E1 -9215.156,E2 -9215.156} C_VEL
LIN {X 0,Y 439.392,Z 529.748,A -85,B 0,C 180,E1 -9218.594,E2 -9218.594} C_VEL
LIN {X 0,Y 439.386,Z 529.73,A -85,B 0,C 180,E1 -9221.256,E2 -9221.256} C_VEL
LIN {X 0,Y 439.403,Z 529.741,A -85,B 0,C 180,E1 -9224.729,E2 -9224.729} C_VEL
LIN {X 0,Y 439.4,Z 529.746,A -85,B 0,C 180,E1 -9227.795,E2 -9227.795} C_VEL
LIN {X 0,Y 439.393,Z 529.728,A -85,B 0,C 180,E1 -9230.223,E2 -9230.223} C_VEL
LIN {X 0,Y 439.377,Z 529.753,A -85,B 0,C 180,E1 -9233.712,E2 -9233.712} C_VEL
LIN {X 0,Y 439.376,Z 529.757,A -85,B 0,C 180,E1 -9237.054,E2 -9237.054} C_VEL
LIN {X 0,Y 439.387,Z 529.753,A -85,B 0,C 180,E1 -9240.274,E2 -9240.274} C_VEL
LIN {X 0,Y 439.433,Z 529.747,A -85,B 0,C 180,E1 -9243.396,E2 -9243.396} C_VEL
LIN {X 0,Y 439.424,Z 529.751,A -85,B 0,C 180,E1 -9246.93,E2 -9246.93} C_VEL
LIN {X 0,Y 439.445,Z 529.943,A -85,B 0,C 180,E1 -9247.242,E2 -9247.242} C_VEL
LIN {X 0,Y 441.174,Z 539.02,A -85,B 0,C 180,E1 -9249.484,E2 -9249.484} C_VEL
LIN {X 0,Y 440.75,Z 549.905,A -85,B 0,C 180,E1 -9251.899,E2 -9251.899} C_VEL
LIN {X 0,Y 441.535,Z 554.077,A -85,B 0,C 180,E1 -9252.048,E2 -9252.048} C_VEL
LIN {X 0,Y 443.431,Z 563.572,A -85,B 0,C 180,E1 -9252.287,E2 -9252.287} C_VEL
LIN {X 0,Y 443.24,Z 567.471,A -85,B 0,C 180,E1 -9252.344,E2 -9252.344} C_VEL
LIN {X 0,Y 440.801,Z 573.725,A -85,B 0,C 180,E1 -9252.347,E2 -9252.347} C_VEL
LIN {X 0,Y 438.037,Z 580.006,A -85,B 0,C 180,E1 -9252.336,E2 -9252.336} C_VEL
LIN {X 0,Y 437.382,Z 583.982,A -85,B 0,C 180,E1 -9252.376,E2 -9252.376} C_VEL
LIN {X 0,Y 436.576,Z 657.385,A -85,B 0,C 180,E1 -9253.607,E2 -9253.607} C_VEL
LIN {X 0,Y 436.184,Z 671.242,A -85,B 0,C 180,E1 -9254.042,E2 -9254.042} C_VEL
LIN {X 0,Y 435.667,Z 683.636,A -85,B 0,C 180,E1 -9254.623,E2 -9254.623} C_VEL
LIN {X 0,Y 435.064,Z 695.48,A -85,B 0,C 180,E1 -9255.38,E2 -9255.38} C_VEL
LIN {X 0,Y 434.474,Z 707.333,A -85,B 0,C 180,E1 -9256.361,E2 -9256.361} C_VEL
LIN {X 0,Y 433.848,Z 717.076,A -85,B 0,C 180,E1 -9257.367,E2 -9257.367} C_VEL
LIN {X 0,Y 433.186,Z 726.26,A -85,B 0,C 180,E1 -9258.536,E2 -9258.536} C_VEL
LIN {X 0,Y 432.557,Z 735.177,A -85,B 0,C 180,E1 -9259.94,E2 -9259.94} C_VEL
LIN {X 0,Y 432.091,Z 742.353,A -85,B 0,C 180,E1 -9261.346,E2 -9261.346} C_VEL
LIN {X 0,Y 431.736,Z 747.197,A -85,B 0,C 180,E1 -9262.517,E2 -9262.517} C_VEL
LIN {X 0,Y 431.617,Z 751.896,A -85,B 0,C 180,E1 -9263.924,E2 -9263.924} C_VEL
LIN {X 0,Y 431.352,Z 755.496,A -85,B 0,C 180,E1 -9265.326,E2 -9265.326} C_VEL
LIN {X 0,Y 431.333,Z 757.354,A -85,B 0,C 180,E1 -9266.262,E2 -9266.262} C_VEL
LIN {X 0,Y 431.326,Z 758.755,A -85,B 0,C 180,E1 -9267.197,E2 -9267.197} C_VEL
LIN {X 0,Y 431.172,Z 760.372,A -85,B 0,C 180,E1 -9269.065,E2 -9269.065} C_VEL
LIN {X 0,Y 431.168,Z 760.607,A -85,B 0,C 180,E1 -9269.999,E2 -9269.999} C_VEL
LIN {X 0,Y 431.172,Z 760.42,A -85,B 0,C 180,E1 -9270.933,E2 -9270.933} C_VEL
LIN {X 0,Y 431.324,Z 758.871,A -85,B 0,C 180,E1 -9272.801,E2 -9272.801} C_VEL
LIN {X 0,Y 431.318,Z 757.518,A -85,B 0,C 180,E1 -9273.736,E2 -9273.736} C_VEL
LIN {X 0,Y 431.427,Z 754.653,A -85,B 0,C 180,E1 -9275.14,E2 -9275.14} C_VEL
LIN {X 0,Y 431.64,Z 750.344,A -85,B 0,C 180,E1 -9276.68,E2 -9276.68} C_VEL
LIN {X 0,Y 431.871,Z 745.758,A -85,B 0,C 180,E1 -9277.95,E2 -9277.95} C_VEL
LIN {X 0,Y 432.311,Z 739.45,A -85,B 0,C 180,E1 -9279.355,E2 -9279.355} C_VEL
LIN {X 0,Y 432.839,Z 731.55,A -85,B 0,C 180,E1 -9280.761,E2 -9280.761} C_VEL
LIN {X 0,Y 433.323,Z 723.5,A -85,B 0,C 180,E1 -9281.933,E2 -9281.933} C_VEL
LIN {X 0,Y 434.092,Z 713.668,A -85,B 0,C 180,E1 -9283.1,E2 -9283.1} C_VEL
LIN {X 0,Y 434.672,Z 702.622,A -85,B 0,C 180,E1 -9284.154,E2 -9284.154} C_VEL
LIN {X 0,Y 435.295,Z 691.781,A -85,B 0,C 180,E1 -9284.97,E2 -9284.97} C_VEL
LIN {X 0,Y 435.883,Z 679.8,A -85,B 0,C 180,E1 -9285.667,E2 -9285.667} C_VEL
LIN {X 0,Y 436.316,Z 666.661,A -85,B 0,C 180,E1 -9286.221,E2 -9286.221} C_VEL
LIN {X 0,Y 436.731,Z 654.945,A -85,B 0,C 180,E1 -9286.536,E2 -9286.536} C_VEL
LIN {X 0,Y 437.389,Z 568.129,A -85,B 0,C 180,E1 -9287.986,E2 -9287.986} C_VEL
LIN {X 0,Y 433.874,Z 550.52,A -85,B 0,C 180,E1 -9288.461,E2 -9288.461} C_VEL
LIN {X 0,Y 433.83,Z 549.071,A -85,B 0,C 180,E1 -9288.683,E2 -9288.683} C_VEL
LIN {X 0,Y 434.243,Z 541.496,A -85,B 0,C 180,E1 -9290.419,E2 -9290.419} C_VEL
LIN {X 0,Y 432.851,Z 532.983,A -85,B 0,C 180,E1 -9292.511,E2 -9292.511} C_VEL
LIN {X 0,Y 432.397,Z 530.646,A -85,B 0,C 180,E1 -9293.18,E2 -9293.18} C_VEL
LIN {X 0,Y 432.399,Z 530.618,A -85,B 0,C 180,E1 -9296.627,E2 -9296.627} C_VEL
LIN {X 0,Y 432.342,Z 530.621,A -85,B 0,C 180,E1 -9299.186,E2 -9299.186} C_VEL
LIN {X 0,Y 432.321,Z 530.63,A -85,B 0,C 180,E1 -9302.442,E2 -9302.442} C_VEL
LIN {X 0,Y 432.343,Z 530.627,A -85,B 0,C 180,E1 -9305.631,E2 -9305.631} C_VEL
LIN {X 0,Y 432.35,Z 530.627,A -85,B 0,C 180,E1 -9308.716,E2 -9308.716} C_VEL
LIN {X 0,Y 432.332,Z 530.632,A -85,B 0,C 180,E1 -9311.796,E2 -9311.796} C_VEL
LIN {X 0,Y 432.336,Z 530.62,A -85,B 0,C 180,E1 -9314.345,E2 -9314.345} C_VEL
LIN {X 0,Y 432.316,Z 530.63,A -85,B 0,C 180,E1 -9317.015,E2 -9317.015} C_VEL
LIN {X 0,Y 432.352,Z 530.62,A -85,B 0,C 180,E1 -9319.816,E2 -9319.816} C_VEL
LIN {X 0,Y 432.312,Z 530.624,A -85,B 0,C 180,E1 -9323.022,E2 -9323.022} C_VEL
LIN {X 0,Y 432.357,Z 530.626,A -85,B 0,C 180,E1 -9325.995,E2 -9325.995} C_VEL
LIN {X 0,Y 432.389,Z 530.625,A -85,B 0,C 180,E1 -9329.743,E2 -9329.743} C_VEL
LIN {X 0,Y 432.394,Z 530.621,A -85,B 0,C 180,E1 -9333.372,E2 -9333.372} C_VEL
LIN {X 0,Y 432.365,Z 530.624,A -85,B 0,C 180,E1 -9336.023,E2 -9336.023} C_VEL
LIN {X 0,Y 432.343,Z 530.624,A -85,B 0,C 180,E1 -9339.046,E2 -9339.046} C_VEL
LIN {X 0,Y 432.371,Z 530.622,A -85,B 0,C 180,E1 -9342.011,E2 -9342.011} C_VEL
LIN {X 0,Y 432.388,Z 530.617,A -85,B 0,C 180,E1 -9344.926,E2 -9344.926} C_VEL
LIN {X 0,Y 432.451,Z 530.615,A -85,B 0,C 180,E1 -9347.803,E2 -9347.803} C_VEL
LIN {X 0,Y 432.484,Z 530.61,A -85,B 0,C 180,E1 -9351.59,E2 -9351.59} C_VEL
LIN {X 0,Y 432.591,Z 530.595,A -85,B 0,C 180,E1 -9354.406,E2 -9354.406} C_VEL
LIN {X 0,Y 432.598,Z 530.594,A -85,B 0,C 180,E1 -9358.138,E2 -9358.138} C_VEL
LIN {X 0,Y 432.727,Z 530.581,A -85,B 0,C 180,E1 -9360,E2 -9360} C_VEL
LIN {X 0,Y 432.599,Z 530.591,A -85,B 0,C 180,E1 -9362.794,E2 -9362.794} C_VEL
LIN {X 0,Y 432.565,Z 530.599,A -85,B 0,C 180,E1 -9366.53,E2 -9366.53} C_VEL
LIN {X 0,Y 432.437,Z 530.616,A -85,B 0,C 180,E1 -9369.353,E2 -9369.353} C_VEL
LIN {X 0,Y 432.437,Z 530.615,A -85,B 0,C 180,E1 -9372.812,E2 -9372.812} C_VEL
LIN {X 0,Y 432.405,Z 530.613,A -85,B 0,C 180,E1 -9376.479,E2 -9376.479} C_VEL
LIN {X 0,Y 432.366,Z 530.625,A -85,B 0,C 180,E1 -9379.959,E2 -9379.959} C_VEL
LIN {X 0,Y 432.313,Z 530.629,A -85,B 0,C 180,E1 -9382.965,E2 -9382.965} C_VEL
LIN {X 0,Y 432.358,Z 530.622,A -85,B 0,C 180,E1 -9386.033,E2 -9386.033} C_VEL
LIN {X 0,Y 432.337,Z 530.63,A -85,B 0,C 180,E1 -9389.188,E2 -9389.188} C_VEL
LIN {X 0,Y 432.321,Z 530.63,A -85,B 0,C 180,E1 -9392.443,E2 -9392.443} C_VEL
LIN {X 0,Y 432.34,Z 530.621,A -85,B 0,C 180,E1 -9395.633,E2 -9395.633} C_VEL
LIN {X 0,Y 432.347,Z 530.625,A -85,B 0,C 180,E1 -9398.717,E2 -9398.717} C_VEL
LIN {X 0,Y 432.328,Z 530.625,A -85,B 0,C 180,E1 -9401.798,E2 -9401.798} C_VEL
LIN {X 0,Y 432.374,Z 530.627,A -85,B 0,C 180,E1 -9405.659,E2 -9405.659} C_VEL
LIN {X 0,Y 432.369,Z 530.625,A -85,B 0,C 180,E1 -9408.393,E2 -9408.393} C_VEL
LIN {X 0,Y 432.349,Z 530.612,A -85,B 0,C 180,E1 -9411.853,E2 -9411.853} C_VEL
LIN {X 0,Y 432.338,Z 530.633,A -85,B 0,C 180,E1 -9415.324,E2 -9415.324} C_VEL
LIN {X 0,Y 432.319,Z 530.584,A -85,B 0,C 180,E1 -9418.655,E2 -9418.655} C_VEL
LIN {X 0,Y 432.382,Z 530.626,A -85,B 0,C 180,E1 -9421.878,E2 -9421.878} C_VEL
LIN {X 0,Y 432.429,Z 530.806,A -85,B 0,C 180,E1 -9423.06,E2 -9423.06} C_VEL
LIN {X 0,Y 434.818,Z 542.801,A -85,B 0,C 180,E1 -9425.661,E2 -9425.661} C_VEL
LIN {X 0,Y 435.207,Z 546.733,A -85,B 0,C 180,E1 -9426.468,E2 -9426.468} C_VEL
LIN {X 0,Y 434.18,Z 562.769,A -85,B 0,C 180,E1 -9429.591,E2 -9429.591} C_VEL
LIN {X 0,Y 433.659,Z 573.091,A -85,B 0,C 180,E1 -9431.546,E2 -9431.546} C_VEL
LIN {X 0,Y 437.331,Z 596.391,A -85,B 0,C 180,E1 -9432.128,E2 -9432.128} C_VEL
LIN {X 0,Y 436.478,Z 681.146,A -85,B 0,C 180,E1 -9433.544,E2 -9433.544} C_VEL
LIN {X 0,Y 436.004,Z 694.387,A -85,B 0,C 180,E1 -9433.947,E2 -9433.947} C_VEL
LIN {X 0,Y 435.446,Z 706.541,A -85,B 0,C 180,E1 -9434.496,E2 -9434.496} C_VEL
LIN {X 0,Y 434.794,Z 718.815,A -85,B 0,C 180,E1 -9435.252,E2 -9435.252} C_VEL
LIN {X 0,Y 434.108,Z 729.885,A -85,B 0,C 180,E1 -9436.137,E2 -9436.137} C_VEL
LIN {X 0,Y 433.481,Z 740.852,A -85,B 0,C 180,E1 -9437.239,E2 -9437.239} C_VEL
LIN {X 0,Y 432.896,Z 749.391,A -85,B 0,C 180,E1 -9438.292,E2 -9438.292} C_VEL
LIN {X 0,Y 432.35,Z 757.268,A -85,B 0,C 180,E1 -9439.464,E2 -9439.464} C_VEL
LIN {X 0,Y 431.878,Z 764.966,A -85,B 0,C 180,E1 -9440.872,E2 -9440.872} C_VEL
LIN {X 0,Y 431.535,Z 772.063,A -85,B 0,C 180,E1 -9442.515,E2 -9442.515} C_VEL
LIN {X 0,Y 431.293,Z 777.052,A -85,B 0,C 180,E1 -9444.008,E2 -9444.008} C_VEL
LIN {X 0,Y 431.276,Z 780.399,A -85,B 0,C 180,E1 -9445.327,E2 -9445.327} C_VEL
LIN {X 0,Y 431.189,Z 782.26,A -85,B 0,C 180,E1 -9446.263,E2 -9446.263} C_VEL
LIN {X 0,Y 431.236,Z 783.658,A -85,B 0,C 180,E1 -9447.198,E2 -9447.198} C_VEL
LIN {X 0,Y 431.202,Z 784.652,A -85,B 0,C 180,E1 -9448.133,E2 -9448.133} C_VEL
LIN {X 0,Y 431.167,Z 785.473,A -85,B 0,C 180,E1 -9450.001,E2 -9450.001} C_VEL
LIN {X 0,Y 431.203,Z 784.647,A -85,B 0,C 180,E1 -9451.869,E2 -9451.869} C_VEL
LIN {X 0,Y 431.236,Z 783.65,A -85,B 0,C 180,E1 -9452.803,E2 -9452.803} C_VEL
LIN {X 0,Y 431.19,Z 782.25,A -85,B 0,C 180,E1 -9453.739,E2 -9453.739} C_VEL
LIN {X 0,Y 431.304,Z 779.316,A -85,B 0,C 180,E1 -9455.143,E2 -9455.143} C_VEL
LIN {X 0,Y 431.378,Z 775.341,A -85,B 0,C 180,E1 -9456.549,E2 -9456.549} C_VEL
LIN {X 0,Y 431.681,Z 769.226,A -85,B 0,C 180,E1 -9458.191,E2 -9458.191} C_VEL
LIN {X 0,Y 432.013,Z 762.545,A -85,B 0,C 180,E1 -9459.599,E2 -9459.599} C_VEL
LIN {X 0,Y 432.527,Z 754.259,A -85,B 0,C 180,E1 -9461.007,E2 -9461.007} C_VEL
LIN {X 0,Y 433.142,Z 745.769,A -85,B 0,C 180,E1 -9462.178,E2 -9462.178} C_VEL
LIN {X 0,Y 433.714,Z 736.06,A -85,B 0,C 180,E1 -9463.272,E2 -9463.272} C_VEL
LIN {X 0,Y 434.387,Z 724.892,A -85,B 0,C 180,E1 -9464.285,E2 -9464.285} C_VEL
LIN {X 0,Y 435.067,Z 713.519,A -85,B 0,C 180,E1 -9465.099,E2 -9465.099} C_VEL
LIN {X 0,Y 435.705,Z 701.85,A -85,B 0,C 180,E1 -9465.736,E2 -9465.736} C_VEL
LIN {X 0,Y 436.217,Z 688.387,A -85,B 0,C 180,E1 -9466.257,E2 -9466.257} C_VEL
LIN {X 0,Y 436.589,Z 675.05,A -85,B 0,C 180,E1 -9466.573,E2 -9466.573} C_VEL
LIN {X 0,Y 437.148,Z 595.14,A -85,B 0,C 180,E1 -9467.897,E2 -9467.897} C_VEL
LIN {X 0,Y 433.664,Z 573.258,A -85,B 0,C 180,E1 -9468.435,E2 -9468.435} C_VEL
LIN {X 0,Y 433.824,Z 569.219,A -85,B 0,C 180,E1 -9469.151,E2 -9469.151} C_VEL
LIN {X 0,Y 435.037,Z 549.664,A -85,B 0,C 180,E1 -9472.952,E2 -9472.952} C_VEL
LIN {X 0,Y 435.188,Z 545.303,A -85,B 0,C 180,E1 -9473.812,E2 -9473.812} C_VEL
LIN {X 0,Y 433.347,Z 535.13,A -85,B 0,C 180,E1 -9475.97,E2 -9475.97} C_VEL
LIN {X 0,Y 432.457,Z 530.673,A -85,B 0,C 180,E1 -9477.004,E2 -9477.004} C_VEL
LIN {X 0,Y 432.351,Z 530.628,A -85,B 0,C 180,E1 -9480.511,E2 -9480.511} C_VEL
LIN {X 0,Y 432.363,Z 530.629,A -85,B 0,C 180,E1 -9484.004,E2 -9484.004} C_VEL
LIN {X 0,Y 432.326,Z 530.631,A -85,B 0,C 180,E1 -9487.197,E2 -9487.197} C_VEL
LIN {X 0,Y 432.337,Z 530.632,A -85,B 0,C 180,E1 -9490.179,E2 -9490.179} C_VEL
LIN {X 0,Y 432.321,Z 530.633,A -85,B 0,C 180,E1 -9493.061,E2 -9493.061} C_VEL
LIN {X 0,Y 432.336,Z 530.632,A -85,B 0,C 180,E1 -9495.665,E2 -9495.665} C_VEL
LIN {X 0,Y 432.337,Z 530.634,A -85,B 0,C 180,E1 -9498.398,E2 -9498.398} C_VEL
LIN {X 0,Y 432.351,Z 530.632,A -85,B 0,C 180,E1 -9501.851,E2 -9501.851} C_VEL
LIN {X 0,Y 432.344,Z 530.63,A -85,B 0,C 180,E1 -9505.323,E2 -9505.323} C_VEL
LIN {X 0,Y 432.325,Z 530.635,A -85,B 0,C 180,E1 -9508.654,E2 -9508.654} C_VEL
LIN {X 0,Y 432.429,Z 530.812,A -85,B 0,C 180,E1 -9511.534,E2 -9511.534} C_VEL
LIN {X 0,Y 434.905,Z 540.928,A -85,B 0,C 180,E1 -9513.357,E2 -9513.357} C_VEL
LIN {X 0,Y 435.93,Z 547.916,A -85,B 0,C 180,E1 -9514.533,E2 -9514.533} C_VEL
LIN {X 0,Y 435.176,Z 568.054,A -85,B 0,C 180,E1 -9517.696,E2 -9517.696} C_VEL
LIN {X 0,Y 434.287,Z 589.902,A -85,B 0,C 180,E1 -9521.116,E2 -9521.116} C_VEL
LIN {X 0,Y 433.586,Z 611.227,A -85,B 0,C 180,E1 -9524.487,E2 -9524.487} C_VEL
LIN {X 0,Y 433.407,Z 617.135,A -85,B 0,C 180,E1 -9525.368,E2 -9525.368} C_VEL
LIN {X 0,Y 435.306,Z 631.663,A -85,B 0,C 180,E1 -9525.768,E2 -9525.768} C_VEL
LIN {X 0,Y 434.352,Z 697.58,A -85,B 0,C 180,E1 -9527.115,E2 -9527.115} C_VEL
LIN {X 0,Y 434.075,Z 707.793,A -85,B 0,C 180,E1 -9527.464,E2 -9527.464} C_VEL
LIN {X 0,Y 433.771,Z 717.966,A -85,B 0,C 180,E1 -9527.96,E2 -9527.96} C_VEL
LIN {X 0,Y 433.379,Z 728.599,A -85,B 0,C 180,E1 -9528.66,E2 -9528.66} C_VEL
LIN {X 0,Y 432.941,Z 737.973,A -85,B 0,C 180,E1 -9529.477,E2 -9529.477} C_VEL
LIN {X 0,Y 432.639,Z 744.6,A -85,B 0,C 180,E1 -9530.179,E2 -9530.179} C_VEL
LIN {X 0,Y 432.224,Z 751.925,A -85,B 0,C 180,E1 -9531.114,E2 -9531.114} C_VEL
LIN {X 0,Y 431.91,Z 757.966,A -85,B 0,C 180,E1 -9532.05,E2 -9532.05} C_VEL
LIN {X 0,Y 431.707,Z 764.262,A -85,B 0,C 180,E1 -9533.245,E2 -9533.245} C_VEL
LIN {X 0,Y 431.55,Z 769.018,A -85,B 0,C 180,E1 -9534.393,E2 -9534.393} C_VEL
LIN {X 0,Y 431.3,Z 773.333,A -85,B 0,C 180,E1 -9535.795,E2 -9535.795} C_VEL
LIN {X 0,Y 431.292,Z 776.321,A -85,B 0,C 180,E1 -9537.198,E2 -9537.198} C_VEL
LIN {X 0,Y 431.205,Z 777.624,A -85,B 0,C 180,E1 -9538.132,E2 -9538.132} C_VEL
LIN {X 0,Y 431.148,Z 778.415,A -85,B 0,C 180,E1 -9539.066,E2 -9539.066} C_VEL
LIN {X 0,Y 431.143,Z 778.69,A -85,B 0,C 180,E1 -9540,E2 -9540} C_VEL
LIN {X 0,Y 431.148,Z 778.371,A -85,B 0,C 180,E1 -9540.934,E2 -9540.934} C_VEL
LIN {X 0,Y 431.205,Z 777.503,A -85,B 0,C 180,E1 -9541.868,E2 -9541.868} C_VEL
LIN {X 0,Y 431.26,Z 776.122,A -85,B 0,C 180,E1 -9542.802,E2 -9542.802} C_VEL
LIN {X 0,Y 431.285,Z 773.036,A -85,B 0,C 180,E1 -9544.205,E2 -9544.205} C_VEL
LIN {X 0,Y 431.478,Z 768.558,A -85,B 0,C 180,E1 -9545.608,E2 -9545.608} C_VEL
LIN {X 0,Y 431.638,Z 763.575,A -85,B 0,C 180,E1 -9546.773,E2 -9546.773} C_VEL
LIN {X 0,Y 431.775,Z 758.636,A -85,B 0,C 180,E1 -9547.717,E2 -9547.717} C_VEL
LIN {X 0,Y 432.052,Z 752.709,A -85,B 0,C 180,E1 -9548.654,E2 -9548.654} C_VEL
LIN {X 0,Y 432.374,Z 745.518,A -85,B 0,C 180,E1 -9549.591,E2 -9549.591} C_VEL
LIN {X 0,Y 432.761,Z 737.88,A -85,B 0,C 180,E1 -9550.409,E2 -9550.409} C_VEL
LIN {X 0,Y 433.116,Z 728.466,A -85,B 0,C 180,E1 -9551.228,E2 -9551.228} C_VEL
LIN {X 0,Y 433.51,Z 717.758,A -85,B 0,C 180,E1 -9551.929,E2 -9551.929} C_VEL
LIN {X 0,Y 433.791,Z 708.189,A -85,B 0,C 180,E1 -9552.396,E2 -9552.396} C_VEL
LIN {X 0,Y 433.937,Z 699.057,A -85,B 0,C 180,E1 -9552.719,E2 -9552.719} C_VEL
LIN {X 0,Y 434.224,Z 685.833,A -85,B 0,C 180,E1 -9553.007,E2 -9553.007} C_VEL
LIN {X 0,Y 434.692,Z 630.966,A -85,B 0,C 180,E1 -9554.053,E2 -9554.053} C_VEL
LIN {X 0,Y 433.032,Z 616.716,A -85,B 0,C 180,E1 -9554.405,E2 -9554.405} C_VEL
LIN {X 0,Y 433.584,Z 599.191,A -85,B 0,C 180,E1 -9557.182,E2 -9557.182} C_VEL
LIN {X 0,Y 434.457,Z 577.57,A -85,B 0,C 180,E1 -9560.647,E2 -9560.647} C_VEL
LIN {X 0,Y 435.292,Z 556.374,A -85,B 0,C 180,E1 -9564.059,E2 -9564.059} C_VEL
LIN {X 0,Y 435.628,Z 547.218,A -85,B 0,C 180,E1 -9565.537,E2 -9565.537} C_VEL
LIN {X 0,Y 433.553,Z 536.05,A -85,B 0,C 180,E1 -9567.464,E2 -9567.464} C_VEL
LIN {X 0,Y 432.421,Z 530.717,A -85,B 0,C 180,E1 -9568.447,E2 -9568.447} C_VEL
LIN {X 0,Y 432.325,Z 530.635,A -85,B 0,C 180,E1 -9571.346,E2 -9571.346} C_VEL
LIN {X 0,Y 432.344,Z 530.628,A -85,B 0,C 180,E1 -9574.677,E2 -9574.677} C_VEL
LIN {X 0,Y 432.35,Z 530.626,A -85,B 0,C 180,E1 -9578.149,E2 -9578.149} C_VEL
LIN {X 0,Y 432.329,Z 530.603,A -85,B 0,C 180,E1 -9581.601,E2 -9581.601} C_VEL
LIN {X 0,Y 432.337,Z 530.62,A -85,B 0,C 180,E1 -9584.347,E2 -9584.347} C_VEL
LIN {X 0,Y 432.324,Z 530.634,A -85,B 0,C 180,E1 -9587.016,E2 -9587.016} C_VEL
LIN {X 0,Y 432.337,Z 530.608,A -85,B 0,C 180,E1 -9589.821,E2 -9589.821} C_VEL
LIN {X 0,Y 432.31,Z 530.634,A -85,B 0,C 180,E1 -9593.022,E2 -9593.022} C_VEL
LIN {X 0,Y 432.362,Z 530.623,A -85,B 0,C 180,E1 -9595.997,E2 -9595.997} C_VEL
LIN {X 0,Y 432.352,Z 530.631,A -85,B 0,C 180,E1 -9599.489,E2 -9599.489} C_VEL
LIN {X 0,Y 432.395,Z 530.625,A -85,B 0,C 180,E1 -9602.928,E2 -9602.928} C_VEL
LIN {X 0,Y 432.376,Z 530.622,A -85,B 0,C 180,E1 -9606.532,E2 -9606.532} C_VEL
LIN {X 0,Y 432.403,Z 530.882,A -85,B 0,C 180,E1 -9607.04,E2 -9607.04} C_VEL
LIN {X 0,Y 434.043,Z 539.212,A -85,B 0,C 180,E1 -9609.131,E2 -9609.131} C_VEL
LIN {X 0,Y 434.151,Z 543.45,A -85,B 0,C 180,E1 -9610.126,E2 -9610.126} C_VEL
LIN {X 0,Y 433.806,Z 550.174,A -85,B 0,C 180,E1 -9611.608,E2 -9611.608} C_VEL
LIN {X 0,Y 435.262,Z 557.336,A -85,B 0,C 180,E1 -9611.832,E2 -9611.832} C_VEL
LIN {X 0,Y 437.494,Z 569.559,A -85,B 0,C 180,E1 -9612.136,E2 -9612.136} C_VEL
LIN {X 0,Y 437.382,Z 583.982,A -85,B 0,C 180,E1 -9612.376,E2 -9612.376} C_VEL
LIN {X 0,Y 436.746,Z 589.83,A -85,B 0,C 180,E1 -9612.448,E2 -9612.448} C_VEL
LIN {X 0,Y 430.987,Z 608.833,A -85,B 0,C 180,E1 -9612.528,E2 -9612.528} C_VEL
LIN {X 0,Y 430.321,Z 614.683,A -85,B 0,C 180,E1 -9612.6,E2 -9612.6} C_VEL
LIN {X 0,Y 429.777,Z 657.607,A -85,B 0,C 180,E1 -9613.34,E2 -9613.34} C_VEL
LIN {X 0,Y 429.377,Z 671.458,A -85,B 0,C 180,E1 -9613.782,E2 -9613.782} C_VEL
LIN {X 0,Y 428.853,Z 683.848,A -85,B 0,C 180,E1 -9614.372,E2 -9614.372} C_VEL
LIN {X 0,Y 428.194,Z 695.686,A -85,B 0,C 180,E1 -9615.139,E2 -9615.139} C_VEL
LIN {X 0,Y 427.621,Z 706.514,A -85,B 0,C 180,E1 -9616.041,E2 -9616.041} C_VEL
LIN {X 0,Y 426.935,Z 717.284,A -85,B 0,C 180,E1 -9617.159,E2 -9617.159} C_VEL
LIN {X 0,Y 426.207,Z 726.469,A -85,B 0,C 180,E1 -9618.345,E2 -9618.345} C_VEL
LIN {X 0,Y 425.568,Z 735.385,A -85,B 0,C 180,E1 -9619.773,E2 -9619.773} C_VEL
LIN {X 0,Y 425.066,Z 742.56,A -85,B 0,C 180,E1 -9621.202,E2 -9621.202} C_VEL
LIN {X 0,Y 424.684,Z 747.404,A -85,B 0,C 180,E1 -9622.392,E2 -9622.392} C_VEL
LIN {X 0,Y 424.572,Z 751.51,A -85,B 0,C 180,E1 -9623.622,E2 -9623.622} C_VEL
LIN {X 0,Y 424.285,Z 755.702,A -85,B 0,C 180,E1 -9625.248,E2 -9625.248} C_VEL
LIN {X 0,Y 424.239,Z 757.56,A -85,B 0,C 180,E1 -9626.2,E2 -9626.2} C_VEL
LIN {X 0,Y 424.241,Z 758.961,A -85,B 0,C 180,E1 -9627.151,E2 -9627.151} C_VEL
LIN {X 0,Y 424.092,Z 760.576,A -85,B 0,C 180,E1 -9629.05,E2 -9629.05} C_VEL
LIN {X 0,Y 424.085,Z 760.811,A -85,B 0,C 180,E1 -9629.999,E2 -9629.999} C_VEL
LIN {X 0,Y 424.091,Z 760.624,A -85,B 0,C 180,E1 -9630.949,E2 -9630.949} C_VEL
LIN {X 0,Y 424.237,Z 759.075,A -85,B 0,C 180,E1 -9632.848,E2 -9632.848} C_VEL
LIN {X 0,Y 424.225,Z 757.723,A -85,B 0,C 180,E1 -9633.799,E2 -9633.799} C_VEL
LIN {X 0,Y 424.373,Z 754.856,A -85,B 0,C 180,E1 -9635.225,E2 -9635.225} C_VEL
LIN {X 0,Y 424.583,Z 750.827,A -85,B 0,C 180,E1 -9636.701,E2 -9636.701} C_VEL
LIN {X 0,Y 424.818,Z 745.961,A -85,B 0,C 180,E1 -9638.083,E2 -9638.083} C_VEL
LIN {X 0,Y 425.313,Z 739.652,A -85,B 0,C 180,E1 -9639.51,E2 -9639.51} C_VEL
LIN {X 0,Y 425.874,Z 731.752,A -85,B 0,C 180,E1 -9640.939,E2 -9640.939} C_VEL
LIN {X 0,Y 426.385,Z 723.702,A -85,B 0,C 180,E1 -9642.131,E2 -9642.131} C_VEL
LIN {X 0,Y 427.181,Z 713.868,A -85,B 0,C 180,E1 -9643.315,E2 -9643.315} C_VEL
LIN {X 0,Y 427.801,Z 702.821,A -85,B 0,C 180,E1 -9644.386,E2 -9644.386} C_VEL
LIN {X 0,Y 428.457,Z 691.978,A -85,B 0,C 180,E1 -9645.214,E2 -9645.214} C_VEL
LIN {X 0,Y 429.077,Z 679.995,A -85,B 0,C 180,E1 -9645.923,E2 -9645.923} C_VEL
LIN {X 0,Y 429.522,Z 666.852,A -85,B 0,C 180,E1 -9646.485,E2 -9646.485} C_VEL
LIN {X 0,Y 429.973,Z 653.623,A -85,B 0,C 180,E1 -9646.834,E2 -9646.834} C_VEL
LIN {X 0,Y 430.671,Z 569.305,A -85,B 0,C 180,E1 -9648.26,E2 -9648.26} C_VEL
LIN {X 0,Y 426.953,Z 550.812,A -85,B 0,C 180,E1 -9648.766,E2 -9648.766} C_VEL
LIN {X 0,Y 426.912,Z 549.85,A -85,B 0,C 180,E1 -9648.881,E2 -9648.881} C_VEL
LIN {X 0,Y 427.227,Z 542.144,A -85,B 0,C 180,E1 -9650.661,E2 -9650.661} C_VEL
LIN {X 0,Y 425.548,Z 532.513,A -85,B 0,C 180,E1 -9653.08,E2 -9653.08} C_VEL
LIN {X 0,Y 425.35,Z 531.52,A -85,B 0,C 180,E1 -9653.426,E2 -9653.426} C_VEL
LIN {X 0,Y 425.347,Z 531.498,A -85,B 0,C 180,E1 -9656.843,E2 -9656.843} C_VEL
LIN {X 0,Y 425.29,Z 531.499,A -85,B 0,C 180,E1 -9659.718,E2 -9659.718} C_VEL
LIN {X 0,Y 425.28,Z 531.508,A -85,B 0,C 180,E1 -9663.047,E2 -9663.047} C_VEL
LIN {X 0,Y 425.282,Z 531.505,A -85,B 0,C 180,E1 -9665.928,E2 -9665.928} C_VEL
LIN {X 0,Y 425.301,Z 531.507,A -85,B 0,C 180,E1 -9669.043,E2 -9669.043} C_VEL
LIN {X 0,Y 425.288,Z 531.508,A -85,B 0,C 180,E1 -9671.958,E2 -9671.958} C_VEL
LIN {X 0,Y 425.282,Z 531.5,A -85,B 0,C 180,E1 -9675.282,E2 -9675.282} C_VEL
LIN {X 0,Y 425.3,Z 531.505,A -85,B 0,C 180,E1 -9678.624,E2 -9678.624} C_VEL
LIN {X 0,Y 425.319,Z 531.492,A -85,B 0,C 180,E1 -9681.103,E2 -9681.103} C_VEL
LIN {X 0,Y 425.298,Z 531.505,A -85,B 0,C 180,E1 -9684.664,E2 -9684.664} C_VEL
LIN {X 0,Y 425.261,Z 531.509,A -85,B 0,C 180,E1 -9688.072,E2 -9688.072} C_VEL
LIN {X 0,Y 425.332,Z 531.503,A -85,B 0,C 180,E1 -9691.368,E2 -9691.368} C_VEL
LIN {X 0,Y 425.289,Z 531.505,A -85,B 0,C 180,E1 -9694.554,E2 -9694.554} C_VEL
LIN {X 0,Y 425.281,Z 531.505,A -85,B 0,C 180,E1 -9697.661,E2 -9697.661} C_VEL
LIN {X 0,Y 425.355,Z 531.497,A -85,B 0,C 180,E1 -9700.704,E2 -9700.704} C_VEL
LIN {X 0,Y 425.381,Z 531.491,A -85,B 0,C 180,E1 -9703.688,E2 -9703.688} C_VEL
LIN {X 0,Y 425.404,Z 531.495,A -85,B 0,C 180,E1 -9707.598,E2 -9707.598} C_VEL
LIN {X 0,Y 425.435,Z 531.486,A -85,B 0,C 180,E1 -9711.45,E2 -9711.45} C_VEL
LIN {X 0,Y 425.547,Z 531.473,A -85,B 0,C 180,E1 -9714.313,E2 -9714.313} C_VEL
LIN {X 0,Y 425.568,Z 531.47,A -85,B 0,C 180,E1 -9718.107,E2 -9718.107} C_VEL
LIN {X 0,Y 425.697,Z 531.457,A -85,B 0,C 180,E1 -9720,E2 -9720} C_VEL
LIN {X 0,Y 425.55,Z 531.469,A -85,B 0,C 180,E1 -9722.84,E2 -9722.84} C_VEL
LIN {X 0,Y 425.566,Z 531.476,A -85,B 0,C 180,E1 -9725.687,E2 -9725.687} C_VEL
LIN {X 0,Y 425.435,Z 531.485,A -85,B 0,C 180,E1 -9728.55,E2 -9728.55} C_VEL
LIN {X 0,Y 425.422,Z 531.488,A -85,B 0,C 180,E1 -9732.401,E2 -9732.401} C_VEL
LIN {X 0,Y 425.381,Z 531.489,A -85,B 0,C 180,E1 -9736.312,E2 -9736.312} C_VEL
LIN {X 0,Y 425.353,Z 531.503,A -85,B 0,C 180,E1 -9739.648,E2 -9739.648} C_VEL
LIN {X 0,Y 425.3,Z 531.506,A -85,B 0,C 180,E1 -9743.366,E2 -9743.366} C_VEL
LIN {X 0,Y 425.342,Z 531.494,A -85,B 0,C 180,E1 -9746.845,E2 -9746.845} C_VEL
LIN {X 0,Y 425.284,Z 531.51,A -85,B 0,C 180,E1 -9749.72,E2 -9749.72} C_VEL
LIN {X 0,Y 425.278,Z 531.508,A -85,B 0,C 180,E1 -9753.048,E2 -9753.048} C_VEL
LIN {X 0,Y 425.279,Z 531.496,A -85,B 0,C 180,E1 -9755.93,E2 -9755.93} C_VEL
LIN {X 0,Y 425.298,Z 531.505,A -85,B 0,C 180,E1 -9759.045,E2 -9759.045} C_VEL
LIN {X 0,Y 425.269,Z 531.499,A -85,B 0,C 180,E1 -9762.654,E2 -9762.654} C_VEL
LIN {X 0,Y 425.314,Z 531.501,A -85,B 0,C 180,E1 -9766.053,E2 -9766.053} C_VEL
LIN {X 0,Y 425.306,Z 531.505,A -85,B 0,C 180,E1 -9768.627,E2 -9768.627} C_VEL
LIN {X 0,Y 425.32,Z 531.495,A -85,B 0,C 180,E1 -9771.105,E2 -9771.105} C_VEL
LIN {X 0,Y 425.298,Z 531.507,A -85,B 0,C 180,E1 -9774.665,E2 -9774.665} C_VEL
LIN {X 0,Y 425.262,Z 531.465,A -85,B 0,C 180,E1 -9778.074,E2 -9778.074} C_VEL
LIN {X 0,Y 425.33,Z 531.504,A -85,B 0,C 180,E1 -9781.369,E2 -9781.369} C_VEL
LIN {X 0,Y 425.366,Z 531.545,A -85,B 0,C 180,E1 -9782.734,E2 -9782.734} C_VEL
LIN {X 0,Y 427.366,Z 541.365,A -85,B 0,C 180,E1 -9784.953,E2 -9784.953} C_VEL
LIN {X 0,Y 428.284,Z 547.687,A -85,B 0,C 180,E1 -9786.296,E2 -9786.296} C_VEL
LIN {X 0,Y 427.271,Z 562.799,A -85,B 0,C 180,E1 -9789.291,E2 -9789.291} C_VEL
LIN {X 0,Y 426.71,Z 572.905,A -85,B 0,C 180,E1 -9791.236,E2 -9791.236} C_VEL
LIN {X 0,Y 430.556,Z 597.057,A -85,B 0,C 180,E1 -9791.852,E2 -9791.852} C_VEL
LIN {X 0,Y 429.688,Z 680.953,A -85,B 0,C 180,E1 -9793.277,E2 -9793.277} C_VEL
LIN {X 0,Y 429.197,Z 694.19,A -85,B 0,C 180,E1 -9793.685,E2 -9793.685} C_VEL
LIN {X 0,Y 428.619,Z 706.342,A -85,B 0,C 180,E1 -9794.243,E2 -9794.243} C_VEL
LIN {X 0,Y 427.919,Z 718.614,A -85,B 0,C 180,E1 -9795.01,E2 -9795.01} C_VEL
LIN {X 0,Y 427.204,Z 729.554,A -85,B 0,C 180,E1 -9795.896,E2 -9795.896} C_VEL
LIN {X 0,Y 426.503,Z 740.648,A -85,B 0,C 180,E1 -9797.027,E2 -9797.027} C_VEL
LIN {X 0,Y 425.907,Z 749.187,A -85,B 0,C 180,E1 -9798.097,E2 -9798.097} C_VEL
LIN {X 0,Y 425.319,Z 757.064,A -85,B 0,C 180,E1 -9799.288,E2 -9799.288} C_VEL
LIN {X 0,Y 424.834,Z 764.762,A -85,B 0,C 180,E1 -9800.719,E2 -9800.719} C_VEL
LIN {X 0,Y 424.452,Z 771.858,A -85,B 0,C 180,E1 -9802.389,E2 -9802.389} C_VEL
LIN {X 0,Y 424.247,Z 776.207,A -85,B 0,C 180,E1 -9803.695,E2 -9803.695} C_VEL
LIN {X 0,Y 424.205,Z 780.195,A -85,B 0,C 180,E1 -9805.249,E2 -9805.249} C_VEL
LIN {X 0,Y 424.101,Z 782.056,A -85,B 0,C 180,E1 -9806.2,E2 -9806.2} C_VEL
LIN {X 0,Y 424.132,Z 783.453,A -85,B 0,C 180,E1 -9807.151,E2 -9807.151} C_VEL
LIN {X 0,Y 424.128,Z 784.448,A -85,B 0,C 180,E1 -9808.102,E2 -9808.102} C_VEL
LIN {X 0,Y 424.084,Z 785.269,A -85,B 0,C 180,E1 -9810.001,E2 -9810.001} C_VEL
LIN {X 0,Y 424.088,Z 785.067,A -85,B 0,C 180,E1 -9810.95,E2 -9810.95} C_VEL
LIN {X 0,Y 424.129,Z 784.449,A -85,B 0,C 180,E1 -9811.9,E2 -9811.9} C_VEL
LIN {X 0,Y 424.132,Z 783.445,A -85,B 0,C 180,E1 -9812.85,E2 -9812.85} C_VEL
LIN {X 0,Y 424.101,Z 782.045,A -85,B 0,C 180,E1 -9813.801,E2 -9813.801} C_VEL
LIN {X 0,Y 424.217,Z 779.11,A -85,B 0,C 180,E1 -9815.229,E2 -9815.229} C_VEL
LIN {X 0,Y 424.303,Z 775.135,A -85,B 0,C 180,E1 -9816.659,E2 -9816.659} C_VEL
LIN {X 0,Y 424.615,Z 769.019,A -85,B 0,C 180,E1 -9818.328,E2 -9818.328} C_VEL
LIN {X 0,Y 424.967,Z 762.338,A -85,B 0,C 180,E1 -9819.76,E2 -9819.76} C_VEL
LIN {X 0,Y 425.509,Z 754.051,A -85,B 0,C 180,E1 -9821.191,E2 -9821.191} C_VEL
LIN {X 0,Y 426.171,Z 745.561,A -85,B 0,C 180,E1 -9822.38,E2 -9822.38} C_VEL
LIN {X 0,Y 426.84,Z 735.147,A -85,B 0,C 180,E1 -9823.562,E2 -9823.562} C_VEL
LIN {X 0,Y 427.482,Z 724.683,A -85,B 0,C 180,E1 -9824.521,E2 -9824.521} C_VEL
LIN {X 0,Y 428.211,Z 713.31,A -85,B 0,C 180,E1 -9825.347,E2 -9825.347} C_VEL
LIN {X 0,Y 428.865,Z 701.639,A -85,B 0,C 180,E1 -9825.993,E2 -9825.993} C_VEL
LIN {X 0,Y 429.408,Z 688.173,A -85,B 0,C 180,E1 -9826.522,E2 -9826.522} C_VEL
LIN {X 0,Y 429.8,Z 674.829,A -85,B 0,C 180,E1 -9826.843,E2 -9826.843} C_VEL
LIN {X 0,Y 430.416,Z 596.225,A -85,B 0,C 180,E1 -9828.164,E2 -9828.164} C_VEL
LIN {X 0,Y 426.735,Z 573.062,A -85,B 0,C 180,E1 -9828.744,E2 -9828.744} C_VEL
LIN {X 0,Y 426.918,Z 569.016,A -85,B 0,C 180,E1 -9829.473,E2 -9829.473} C_VEL
LIN {X 0,Y 428.135,Z 550.172,A -85,B 0,C 180,E1 -9833.202,E2 -9833.202} C_VEL
LIN {X 0,Y 428.237,Z 546.38,A -85,B 0,C 180,E1 -9833.966,E2 -9833.966} C_VEL
LIN {X 0,Y 426.076,Z 534.942,A -85,B 0,C 180,E1 -9836.447,E2 -9836.447} C_VEL
LIN {X 0,Y 425.374,Z 531.549,A -85,B 0,C 180,E1 -9837.27,E2 -9837.27} C_VEL
LIN {X 0,Y 425.294,Z 531.51,A -85,B 0,C 180,E1 -9840.761,E2 -9840.761} C_VEL
LIN {X 0,Y 425.315,Z 531.509,A -85,B 0,C 180,E1 -9844.288,E2 -9844.288} C_VEL
LIN {X 0,Y 425.283,Z 531.51,A -85,B 0,C 180,E1 -9847.695,E2 -9847.695} C_VEL
LIN {X 0,Y 425.283,Z 531.509,A -85,B 0,C 180,E1 -9850.52,E2 -9850.52} C_VEL
LIN {X 0,Y 425.261,Z 531.512,A -85,B 0,C 180,E1 -9853.351,E2 -9853.351} C_VEL
LIN {X 0,Y 425.261,Z 531.515,A -85,B 0,C 180,E1 -9856.649,E2 -9856.649} C_VEL
LIN {X 0,Y 425.298,Z 531.508,A -85,B 0,C 180,E1 -9859.874,E2 -9859.874} C_VEL
LIN {X 0,Y 425.288,Z 531.51,A -85,B 0,C 180,E1 -9862.487,E2 -9862.487} C_VEL
LIN {X 0,Y 425.311,Z 531.509,A -85,B 0,C 180,E1 -9865.818,E2 -9865.818} C_VEL
LIN {X 0,Y 425.294,Z 531.511,A -85,B 0,C 180,E1 -9869.239,E2 -9869.239} C_VEL
LIN {X 0,Y 425.364,Z 531.757,A -85,B 0,C 180,E1 -9871.127,E2 -9871.127} C_VEL
LIN {X 0,Y 428.185,Z 542.878,A -85,B 0,C 180,E1 -9873.184,E2 -9873.184} C_VEL
LIN {X 0,Y 429.17,Z 549.026,A -85,B 0,C 180,E1 -9874.247,E2 -9874.247} C_VEL
LIN {X 0,Y 428.42,Z 568.368,A -85,B 0,C 180,E1 -9877.325,E2 -9877.325} C_VEL
LIN {X 0,Y 427.478,Z 590.243,A -85,B 0,C 180,E1 -9880.803,E2 -9880.803} C_VEL
LIN {X 0,Y 426.699,Z 611.698,A -85,B 0,C 180,E1 -9884.231,E2 -9884.231} C_VEL
LIN {X 0,Y 426.528,Z 617.152,A -85,B 0,C 180,E1 -9885.051,E2 -9885.051} C_VEL
LIN {X 0,Y 428.541,Z 632.383,A -85,B 0,C 180,E1 -9885.497,E2 -9885.497} C_VEL
LIN {X 0,Y 427.508,Z 697.957,A -85,B 0,C 180,E1 -9886.875,E2 -9886.875} C_VEL
LIN {X 0,Y 427.215,Z 707.989,A -85,B 0,C 180,E1 -9887.229,E2 -9887.229} C_VEL
LIN {X 0,Y 426.857,Z 718.595,A -85,B 0,C 180,E1 -9887.762,E2 -9887.762} C_VEL
LIN {X 0,Y 426.441,Z 728.99,A -85,B 0,C 180,E1 -9888.473,E2 -9888.473} C_VEL
LIN {X 0,Y 425.974,Z 738.278,A -85,B 0,C 180,E1 -9889.303,E2 -9889.303} C_VEL
LIN {X 0,Y 425.658,Z 744.847,A -85,B 0,C 180,E1 -9890.017,E2 -9890.017} C_VEL
LIN {X 0,Y 425.225,Z 752.15,A -85,B 0,C 180,E1 -9890.966,E2 -9890.966} C_VEL
LIN {X 0,Y 424.84,Z 759.577,A -85,B 0,C 180,E1 -9892.156,E2 -9892.156} C_VEL
LIN {X 0,Y 424.631,Z 765.406,A -85,B 0,C 180,E1 -9893.347,E2 -9893.347} C_VEL
LIN {X 0,Y 424.5,Z 769.184,A -85,B 0,C 180,E1 -9894.299,E2 -9894.299} C_VEL
LIN {X 0,Y 424.218,Z 773.472,A -85,B 0,C 180,E1 -9895.725,E2 -9895.725} C_VEL
LIN {X 0,Y 424.193,Z 776.443,A -85,B 0,C 180,E1 -9897.151,E2 -9897.151} C_VEL
LIN {X 0,Y 424.133,Z 777.722,A -85,B 0,C 180,E1 -9898.101,E2 -9898.101} C_VEL
LIN {X 0,Y 424.069,Z 778.487,A -85,B 0,C 180,E1 -9899.05,E2 -9899.05} C_VEL
LIN {X 0,Y 424.061,Z 778.74,A -85,B 0,C 180,E1 -9900,E2 -9900} C_VEL
LIN {X 0,Y 424.069,Z 778.41,A -85,B 0,C 180,E1 -9900.95,E2 -9900.95} C_VEL
LIN {X 0,Y 424.132,Z 777.513,A -85,B 0,C 180,E1 -9901.899,E2 -9901.899} C_VEL
LIN {X 0,Y 424.159,Z 776.097,A -85,B 0,C 180,E1 -9902.849,E2 -9902.849} C_VEL
LIN {X 0,Y 424.204,Z 772.972,A -85,B 0,C 180,E1 -9904.276,E2 -9904.276} C_VEL
LIN {X 0,Y 424.387,Z 768.408,A -85,B 0,C 180,E1 -9905.703,E2 -9905.703} C_VEL
LIN {X 0,Y 424.568,Z 763.338,A -85,B 0,C 180,E1 -9906.893,E2 -9906.893} C_VEL
LIN {X 0,Y 424.731,Z 758.366,A -85,B 0,C 180,E1 -9907.846,E2 -9907.846} C_VEL
LIN {X 0,Y 425.006,Z 752.369,A -85,B 0,C 180,E1 -9908.799,E2 -9908.799} C_VEL
LIN {X 0,Y 425.354,Z 745.098,A -85,B 0,C 180,E1 -9909.751,E2 -9909.751} C_VEL
LIN {X 0,Y 425.802,Z 736.18,A -85,B 0,C 180,E1 -9910.701,E2 -9910.701} C_VEL
LIN {X 0,Y 426.239,Z 726.112,A -85,B 0,C 180,E1 -9911.532,E2 -9911.532} C_VEL
LIN {X 0,Y 426.528,Z 716.768,A -85,B 0,C 180,E1 -9912.127,E2 -9912.127} C_VEL
LIN {X 0,Y 426.768,Z 706.892,A -85,B 0,C 180,E1 -9912.603,E2 -9912.603} C_VEL
LIN {X 0,Y 427.093,Z 695.238,A -85,B 0,C 180,E1 -9912.986,E2 -9912.986} C_VEL
LIN {X 0,Y 427.782,Z 631.694,A -85,B 0,C 180,E1 -9914.231,E2 -9914.231} C_VEL
LIN {X 0,Y 426.03,Z 616.802,A -85,B 0,C 180,E1 -9914.601,E2 -9914.601} C_VEL
LIN {X 0,Y 426.645,Z 598.687,A -85,B 0,C 180,E1 -9917.495,E2 -9917.495} C_VEL
LIN {X 0,Y 427.521,Z 577.419,A -85,B 0,C 180,E1 -9920.937,E2 -9920.937} C_VEL
LIN {X 0,Y 428.364,Z 557.253,A -85,B 0,C 180,E1 -9924.215,E2 -9924.215} C_VEL
LIN {X 0,Y 428.687,Z 548.642,A -85,B 0,C 180,E1 -9925.619,E2 -9925.619} C_VEL
LIN {X 0,Y 426.405,Z 536.441,A -85,B 0,C 180,E1 -9927.75,E2 -9927.75} C_VEL
LIN {X 0,Y 425.35,Z 531.587,A -85,B 0,C 180,E1 -9928.666,E2 -9928.666} C_VEL
LIN {X 0,Y 425.269,Z 531.515,A -85,B 0,C 180,E1 -9931.927,E2 -9931.927} C_VEL
LIN {X 0,Y 425.304,Z 531.509,A -85,B 0,C 180,E1 -9935.336,E2 -9935.336} C_VEL
LIN {X 0,Y 425.304,Z 531.505,A -85,B 0,C 180,E1 -9939.044,E2 -9939.044} C_VEL
LIN {X 0,Y 425.274,Z 531.478,A -85,B 0,C 180,E1 -9942.653,E2 -9942.653} C_VEL
LIN {X 0,Y 425.265,Z 531.51,A -85,B 0,C 180,E1 -9946.044,E2 -9946.044} C_VEL
LIN {X 0,Y 425.278,Z 531.504,A -85,B 0,C 180,E1 -9948.621,E2 -9948.621} C_VEL
LIN {X 0,Y 425.296,Z 531.489,A -85,B 0,C 180,E1 -9951.1,E2 -9951.1} C_VEL
LIN {X 0,Y 425.302,Z 531.507,A -85,B 0,C 180,E1 -9954.664,E2 -9954.664} C_VEL
LIN {X 0,Y 425.269,Z 531.509,A -85,B 0,C 180,E1 -9958.073,E2 -9958.073} C_VEL
LIN {X 0,Y 425.336,Z 531.502,A -85,B 0,C 180,E1 -9961.368,E2 -9961.368} C_VEL
LIN {X 0,Y 425.298,Z 531.51,A -85,B 0,C 180,E1 -9964.554,E2 -9964.554} C_VEL
LIN {X 0,Y 425.364,Z 531.64,A -85,B 0,C 180,E1 -9966.764,E2 -9966.764} C_VEL
LIN {X 0,Y 427.195,Z 541.523,A -85,B 0,C 180,E1 -9969.286,E2 -9969.286} C_VEL
LIN {X 0,Y 426.942,Z 549.001,A -85,B 0,C 180,E1 -9971.037,E2 -9971.037} C_VEL
LIN {X 0,Y 426.901,Z 550.631,A -85,B 0,C 180,E1 -9971.321,E2 -9971.321} C_VEL
LIN {X 0,Y 430.737,Z 570.028,A -85,B 0,C 180,E1 -9971.851,E2 -9971.851} C_VEL
LIN {X 0,Y 430.321,Z 614.683,A -85,B 0,C 180,E1 -9972.6,E2 -9972.6} C_VEL
LIN {X 0,Y 429.677,Z 620.528,A -85,B 0,C 180,E1 -9972.673,E2 -9972.673} C_VEL
LIN {X 0,Y 423.968,Z 639.535,A -85,B 0,C 180,E1 -9972.76,E2 -9972.76} C_VEL
LIN {X 0,Y 423.243,Z 645.385,A -85,B 0,C 180,E1 -9972.831,E2 -9972.831} C_VEL
LIN {X 0,Y 422.906,Z 661.246,A -85,B 0,C 180,E1 -9973.154,E2 -9973.154} C_VEL
LIN {X 0,Y 422.533,Z 673.183,A -85,B 0,C 180,E1 -9973.574,E2 -9973.574} C_VEL
LIN {X 0,Y 421.994,Z 685.063,A -85,B 0,C 180,E1 -9974.173,E2 -9974.173} C_VEL
LIN {X 0,Y 421.249,Z 697.474,A -85,B 0,C 180,E1 -9975.012,E2 -9975.012} C_VEL
LIN {X 0,Y 420.627,Z 708.734,A -85,B 0,C 180,E1 -9975.998,E2 -9975.998} C_VEL
LIN {X 0,Y 419.86,Z 719.452,A -85,B 0,C 180,E1 -9977.185,E2 -9977.185} C_VEL
LIN {X 0,Y 419.107,Z 728.297,A -85,B 0,C 180,E1 -9978.39,E2 -9978.39} C_VEL
LIN {X 0,Y 418.469,Z 736.924,A -85,B 0,C 180,E1 -9979.842,E2 -9979.842} C_VEL
LIN {X 0,Y 417.963,Z 743.799,A -85,B 0,C 180,E1 -9981.295,E2 -9981.295} C_VEL
LIN {X 0,Y 417.566,Z 749.305,A -85,B 0,C 180,E1 -9982.747,E2 -9982.747} C_VEL
LIN {X 0,Y 417.412,Z 753.622,A -85,B 0,C 180,E1 -9984.201,E2 -9984.201} C_VEL
LIN {X 0,Y 417.223,Z 755.907,A -85,B 0,C 180,E1 -9985.168,E2 -9985.168} C_VEL
LIN {X 0,Y 417.146,Z 757.766,A -85,B 0,C 180,E1 -9986.135,E2 -9986.135} C_VEL
LIN {X 0,Y 417.158,Z 759.166,A -85,B 0,C 180,E1 -9987.102,E2 -9987.102} C_VEL
LIN {X 0,Y 417.014,Z 760.78,A -85,B 0,C 180,E1 -9989.034,E2 -9989.034} C_VEL
LIN {X 0,Y 417.004,Z 761.015,A -85,B 0,C 180,E1 -9989.999,E2 -9989.999} C_VEL
LIN {X 0,Y 417.014,Z 760.828,A -85,B 0,C 180,E1 -9990.965,E2 -9990.965} C_VEL
LIN {X 0,Y 417.154,Z 759.279,A -85,B 0,C 180,E1 -9992.896,E2 -9992.896} C_VEL
LIN {X 0,Y 417.133,Z 757.927,A -85,B 0,C 180,E1 -9993.863,E2 -9993.863} C_VEL
LIN {X 0,Y 417.32,Z 755.059,A -85,B 0,C 180,E1 -9995.314,E2 -9995.314} C_VEL
LIN {X 0,Y 417.52,Z 751.173,A -85,B 0,C 180,E1 -9996.766,E2 -9996.766} C_VEL
LIN {X 0,Y 417.788,Z 746.164,A -85,B 0,C 180,E1 -9998.22,E2 -9998.22} C_VEL
LIN {X 0,Y 418.31,Z 739.855,A -85,B 0,C 180,E1 -9999.671,E2 -9999.671} C_VEL
LIN {X 0,Y 418.909,Z 731.954,A -85,B 0,C 180,E1 -10001.123,E2 -10001.123} C_VEL
LIN {X 0,Y 419.461,Z 723.903,A -85,B 0,C 180,E1 -10002.334,E2 -10002.334} C_VEL
LIN {X 0,Y 420.287,Z 714.068,A -85,B 0,C 180,E1 -10003.538,E2 -10003.538} C_VEL
LIN {X 0,Y 420.929,Z 703.02,A -85,B 0,C 180,E1 -10004.626,E2 -10004.626} C_VEL
LIN {X 0,Y 421.617,Z 692.176,A -85,B 0,C 180,E1 -10005.467,E2 -10005.467} C_VEL
LIN {X 0,Y 422.28,Z 680.191,A -85,B 0,C 180,E1 -10006.186,E2 -10006.186} C_VEL
LIN {X 0,Y 422.746,Z 667.042,A -85,B 0,C 180,E1 -10006.757,E2 -10006.757} C_VEL
LIN {X 0,Y 423.161,Z 655.308,A -85,B 0,C 180,E1 -10007.082,E2 -10007.082} C_VEL
LIN {X 0,Y 423.928,Z 570.284,A -85,B 0,C 180,E1 -10008.547,E2 -10008.547} C_VEL
LIN {X 0,Y 420.075,Z 550.944,A -85,B 0,C 180,E1 -10009.088,E2 -10009.088} C_VEL
LIN {X 0,Y 420.041,Z 549.552,A -85,B 0,C 180,E1 -10009.301,E2 -10009.301} C_VEL
LIN {X 0,Y 420.265,Z 543.185,A -85,B 0,C 180,E1 -10010.814,E2 -10010.814} C_VEL
LIN {X 0,Y 418.347,Z 532.676,A -85,B 0,C 180,E1 -10013.514,E2 -10013.514} C_VEL
LIN {X 0,Y 418.288,Z 532.377,A -85,B 0,C 180,E1 -10013.78,E2 -10013.78} C_VEL
LIN {X 0,Y 418.309,Z 532.377,A -85,B 0,C 180,E1 -10017.069,E2 -10017.069} C_VEL
LIN {X 0,Y 418.243,Z 532.381,A -85,B 0,C 180,E1 -10020.271,E2 -10020.271} C_VEL
LIN {X 0,Y 418.247,Z 532.389,A -85,B 0,C 180,E1 -10023.676,E2 -10023.676} C_VEL
LIN {X 0,Y 418.243,Z 532.386,A -85,B 0,C 180,E1 -10027.222,E2 -10027.222} C_VEL
LIN {X 0,Y 418.252,Z 532.379,A -85,B 0,C 180,E1 -10029.68,E2 -10029.68} C_VEL
LIN {X 0,Y 418.229,Z 532.386,A -85,B 0,C 180,E1 -10032.321,E2 -10032.321} C_VEL
LIN {X 0,Y 418.234,Z 532.377,A -85,B 0,C 180,E1 -10035.108,E2 -10035.108} C_VEL
LIN {X 0,Y 418.252,Z 532.386,A -85,B 0,C 180,E1 -10037.768,E2 -10037.768} C_VEL
LIN {X 0,Y 418.264,Z 532.372,A -85,B 0,C 180,E1 -10040.616,E2 -10040.616} C_VEL
LIN {X 0,Y 418.243,Z 532.385,A -85,B 0,C 180,E1 -10043.976,E2 -10043.976} C_VEL
LIN {X 0,Y 418.252,Z 532.385,A -85,B 0,C 180,E1 -10047.155,E2 -10047.155} C_VEL
LIN {X 0,Y 418.268,Z 532.381,A -85,B 0,C 180,E1 -10050.838,E2 -10050.838} C_VEL
LIN {X 0,Y 418.264,Z 532.382,A -85,B 0,C 180,E1 -10054.095,E2 -10054.095} C_VEL
LIN {X 0,Y 418.231,Z 532.385,A -85,B 0,C 180,E1 -10057.263,E2 -10057.263} C_VEL
LIN {X 0,Y 418.276,Z 532.379,A -85,B 0,C 180,E1 -10060.364,E2 -10060.364} C_VEL
LIN {X 0,Y 418.31,Z 532.372,A -85,B 0,C 180,E1 -10063.404,E2 -10063.404} C_VEL
LIN {X 0,Y 418.338,Z 532.372,A -85,B 0,C 180,E1 -10066.999,E2 -10066.999} C_VEL
LIN {X 0,Y 418.334,Z 532.364,A -85,B 0,C 180,E1 -10070.328,E2 -10070.328} C_VEL
LIN {X 0,Y 418.486,Z 532.356,A -85,B 0,C 180,E1 -10073.249,E2 -10073.249} C_VEL
LIN {X 0,Y 418.335,Z 532.374,A -85,B 0,C 180,E1 -10075.181,E2 -10075.181} C_VEL
LIN {X 0,Y 418.537,Z 532.346,A -85,B 0,C 180,E1 -10078.075,E2 -10078.075} C_VEL
LIN {X 0,Y 418.667,Z 532.333,A -85,B 0,C 180,E1 -10080,E2 -10080} C_VEL
LIN {X 0,Y 418.504,Z 532.347,A -85,B 0,C 180,E1 -10082.888,E2 -10082.888} C_VEL
LIN {X 0,Y 418.522,Z 532.353,A -85,B 0,C 180,E1 -10085.783,E2 -10085.783} C_VEL
LIN {X 0,Y 418.393,Z 532.362,A -85,B 0,C 180,E1 -10088.695,E2 -10088.695} C_VEL
LIN {X 0,Y 418.324,Z 532.374,A -85,B 0,C 180,E1 -10091.631,E2 -10091.631} C_VEL
LIN {X 0,Y 418.299,Z 532.374,A -85,B 0,C 180,E1 -10094.597,E2 -10094.597} C_VEL
LIN {X 0,Y 418.281,Z 532.38,A -85,B 0,C 180,E1 -10097.604,E2 -10097.604} C_VEL
LIN {X 0,Y 418.253,Z 532.38,A -85,B 0,C 180,E1 -10100.663,E2 -10100.663} C_VEL
LIN {X 0,Y 418.281,Z 532.384,A -85,B 0,C 180,E1 -10103.782,E2 -10103.782} C_VEL
LIN {X 0,Y 418.303,Z 532.372,A -85,B 0,C 180,E1 -10107.071,E2 -10107.071} C_VEL
LIN {X 0,Y 418.238,Z 532.382,A -85,B 0,C 180,E1 -10110.273,E2 -10110.273} C_VEL
LIN {X 0,Y 418.243,Z 532.388,A -85,B 0,C 180,E1 -10113.678,E2 -10113.678} C_VEL
LIN {X 0,Y 418.24,Z 532.372,A -85,B 0,C 180,E1 -10117.224,E2 -10117.224} C_VEL
LIN {X 0,Y 418.25,Z 532.39,A -85,B 0,C 180,E1 -10119.682,E2 -10119.682} C_VEL
LIN {X 0,Y 418.224,Z 532.377,A -85,B 0,C 180,E1 -10122.322,E2 -10122.322} C_VEL
LIN {X 0,Y 418.255,Z 532.384,A -85,B 0,C 180,E1 -10125.113,E2 -10125.113} C_VEL
LIN {X 0,Y 418.289,Z 532.378,A -85,B 0,C 180,E1 -10127.774,E2 -10127.774} C_VEL
LIN {X 0,Y 418.262,Z 532.367,A -85,B 0,C 180,E1 -10131.561,E2 -10131.561} C_VEL
LIN {X 0,Y 418.257,Z 532.386,A -85,B 0,C 180,E1 -10135.16,E2 -10135.16} C_VEL
LIN {X 0,Y 418.243,Z 532.348,A -85,B 0,C 180,E1 -10137.473,E2 -10137.473} C_VEL
LIN {X 0,Y 418.267,Z 532.365,A -85,B 0,C 180,E1 -10140.896,E2 -10140.896} C_VEL
LIN {X 0,Y 418.352,Z 532.554,A -85,B 0,C 180,E1 -10142.528,E2 -10142.528} C_VEL
LIN {X 0,Y 420.855,Z 544.96,A -85,B 0,C 180,E1 -10145.325,E2 -10145.325} C_VEL
LIN {X 0,Y 421.335,Z 548.765,A -85,B 0,C 180,E1 -10146.141,E2 -10146.141} C_VEL
LIN {X 0,Y 420.308,Z 563.854,A -85,B 0,C 180,E1 -10149.188,E2 -10149.188} C_VEL
LIN {X 0,Y 419.802,Z 572.715,A -85,B 0,C 180,E1 -10150.916,E2 -10150.916} C_VEL
LIN {X 0,Y 423.715,Z 597.048,A -85,B 0,C 180,E1 -10151.552,E2 -10151.552} C_VEL
LIN {X 0,Y 422.908,Z 680.76,A -85,B 0,C 180,E1 -10153.001,E2 -10153.001} C_VEL
LIN {X 0,Y 422.391,Z 693.23,A -85,B 0,C 180,E1 -10153.384,E2 -10153.384} C_VEL
LIN {X 0,Y 421.796,Z 706.143,A -85,B 0,C 180,E1 -10153.981,E2 -10153.981} C_VEL
LIN {X 0,Y 421.04,Z 718.413,A -85,B 0,C 180,E1 -10154.759,E2 -10154.759} C_VEL
LIN {X 0,Y 420.27,Z 729.814,A -85,B 0,C 180,E1 -10155.703,E2 -10155.703} C_VEL
LIN {X 0,Y 419.539,Z 740.444,A -85,B 0,C 180,E1 -10156.807,E2 -10156.807} C_VEL
LIN {X 0,Y 418.921,Z 748.984,A -85,B 0,C 180,E1 -10157.896,E2 -10157.896} C_VEL
LIN {X 0,Y 418.316,Z 756.86,A -85,B 0,C 180,E1 -10159.106,E2 -10159.106} C_VEL
LIN {X 0,Y 417.794,Z 764.557,A -85,B 0,C 180,E1 -10160.561,E2 -10160.561} C_VEL
LIN {X 0,Y 417.384,Z 771.653,A -85,B 0,C 180,E1 -10162.259,E2 -10162.259} C_VEL
LIN {X 0,Y 417.146,Z 776.432,A -85,B 0,C 180,E1 -10163.733,E2 -10163.733} C_VEL
LIN {X 0,Y 417.113,Z 779.991,A -85,B 0,C 180,E1 -10165.168,E2 -10165.168} C_VEL
LIN {X 0,Y 417.017,Z 781.852,A -85,B 0,C 180,E1 -10166.135,E2 -10166.135} C_VEL
LIN {X 0,Y 417.029,Z 783.248,A -85,B 0,C 180,E1 -10167.103,E2 -10167.103} C_VEL
LIN {X 0,Y 417.056,Z 784.244,A -85,B 0,C 180,E1 -10168.069,E2 -10168.069} C_VEL
LIN {X 0,Y 417.004,Z 785.194,A -85,B 0,C 180,E1 -10170.001,E2 -10170.001} C_VEL
LIN {X 0,Y 417.01,Z 784.99,A -85,B 0,C 180,E1 -10170.966,E2 -10170.966} C_VEL
LIN {X 0,Y 417.029,Z 783.24,A -85,B 0,C 180,E1 -10172.899,E2 -10172.899} C_VEL
LIN {X 0,Y 417.017,Z 781.84,A -85,B 0,C 180,E1 -10173.866,E2 -10173.866} C_VEL
LIN {X 0,Y 417.132,Z 778.905,A -85,B 0,C 180,E1 -10175.318,E2 -10175.318} C_VEL
LIN {X 0,Y 417.236,Z 774.929,A -85,B 0,C 180,E1 -10176.772,E2 -10176.772} C_VEL
LIN {X 0,Y 417.545,Z 768.812,A -85,B 0,C 180,E1 -10178.47,E2 -10178.47} C_VEL
LIN {X 0,Y 417.946,Z 762.131,A -85,B 0,C 180,E1 -10179.926,E2 -10179.926} C_VEL
LIN {X 0,Y 418.522,Z 753.844,A -85,B 0,C 180,E1 -10181.381,E2 -10181.381} C_VEL
LIN {X 0,Y 419.208,Z 745.353,A -85,B 0,C 180,E1 -10182.589,E2 -10182.589} C_VEL
LIN {X 0,Y 419.911,Z 734.726,A -85,B 0,C 180,E1 -10183.813,E2 -10183.813} C_VEL
LIN {X 0,Y 420.703,Z 723.044,A -85,B 0,C 180,E1 -10184.884,E2 -10184.884} C_VEL
LIN {X 0,Y 421.481,Z 711.174,A -85,B 0,C 180,E1 -10185.722,E2 -10185.722} C_VEL
LIN {X 0,Y 422.139,Z 698.822,A -85,B 0,C 180,E1 -10186.379,E2 -10186.379} C_VEL
LIN {X 0,Y 422.695,Z 686.126,A -85,B 0,C 180,E1 -10186.854,E2 -10186.854} C_VEL
LIN {X 0,Y 423.053,Z 672.82,A -85,B 0,C 180,E1 -10187.151,E2 -10187.151} C_VEL
LIN {X 0,Y 423.695,Z 597.26,A -85,B 0,C 180,E1 -10188.44,E2 -10188.44} C_VEL
LIN {X 0,Y 419.795,Z 572.908,A -85,B 0,C 180,E1 -10189.063,E2 -10189.063} C_VEL
LIN {X 0,Y 419.912,Z 570.068,A -85,B 0,C 180,E1 -10189.557,E2 -10189.557} C_VEL
LIN {X 0,Y 421.232,Z 550.902,A -85,B 0,C 180,E1 -10193.416,E2 -10193.416} C_VEL
LIN {X 0,Y 421.248,Z 547.454,A -85,B 0,C 180,E1 -10194.127,E2 -10194.127} C_VEL
LIN {X 0,Y 419.079,Z 536.014,A -85,B 0,C 180,E1 -10196.655,E2 -10196.655} C_VEL
LIN {X 0,Y 418.347,Z 532.424,A -85,B 0,C 180,E1 -10197.54,E2 -10197.54} C_VEL
LIN {X 0,Y 418.243,Z 532.387,A -85,B 0,C 180,E1 -10201.02,E2 -10201.02} C_VEL
LIN {X 0,Y 418.252,Z 532.384,A -85,B 0,C 180,E1 -10203.677,E2 -10203.677} C_VEL
LIN {X 0,Y 418.244,Z 532.385,A -85,B 0,C 180,E1 -10207.224,E2 -10207.224} C_VEL
LIN {X 0,Y 418.252,Z 532.386,A -85,B 0,C 180,E1 -10209.683,E2 -10209.683} C_VEL
LIN {X 0,Y 418.233,Z 532.388,A -85,B 0,C 180,E1 -10212.321,E2 -10212.321} C_VEL
LIN {X 0,Y 418.239,Z 532.387,A -85,B 0,C 180,E1 -10215.109,E2 -10215.109} C_VEL
LIN {X 0,Y 418.243,Z 532.386,A -85,B 0,C 180,E1 -10217.767,E2 -10217.767} C_VEL
LIN {X 0,Y 418.263,Z 532.384,A -85,B 0,C 180,E1 -10220.618,E2 -10220.618} C_VEL
LIN {X 0,Y 418.249,Z 532.387,A -85,B 0,C 180,E1 -10223.976,E2 -10223.976} C_VEL
LIN {X 0,Y 418.261,Z 532.385,A -85,B 0,C 180,E1 -10227.156,E2 -10227.156} C_VEL
LIN {X 0,Y 418.277,Z 532.578,A -85,B 0,C 180,E1 -10230.639,E2 -10230.639} C_VEL
LIN {X 0,Y 421.286,Z 543.92,A -85,B 0,C 180,E1 -10232.815,E2 -10232.815} C_VEL
LIN {X 0,Y 422.407,Z 550.31,A -85,B 0,C 180,E1 -10233.956,E2 -10233.956} C_VEL
LIN {X 0,Y 421.988,Z 562.377,A -85,B 0,C 180,E1 -10235.919,E2 -10235.919} C_VEL
LIN {X 0,Y 421.031,Z 582.72,A -85,B 0,C 180,E1 -10239.193,E2 -10239.193} C_VEL
LIN {X 0,Y 420.085,Z 605.394,A -85,B 0,C 180,E1 -10242.86,E2 -10242.86} C_VEL
LIN {X 0,Y 419.636,Z 616.997,A -85,B 0,C 180,E1 -10244.705,E2 -10244.705} C_VEL
LIN {X 0,Y 421.688,Z 631.7,A -85,B 0,C 180,E1 -10245.162,E2 -10245.162} C_VEL
LIN {X 0,Y 421.663,Z 642.416,A -85,B 0,C 180,E1 -10245.409,E2 -10245.409} C_VEL
LIN {X 0,Y 420.665,Z 698.335,A -85,B 0,C 180,E1 -10246.627,E2 -10246.627} C_VEL
LIN {X 0,Y 420.359,Z 708.249,A -85,B 0,C 180,E1 -10246.986,E2 -10246.986} C_VEL
LIN {X 0,Y 419.954,Z 719.339,A -85,B 0,C 180,E1 -10247.557,E2 -10247.557} C_VEL
LIN {X 0,Y 419.511,Z 729.504,A -85,B 0,C 180,E1 -10248.28,E2 -10248.28} C_VEL
LIN {X 0,Y 419.099,Z 737.546,A -85,B 0,C 180,E1 -10249.003,E2 -10249.003} C_VEL
LIN {X 0,Y 418.699,Z 745.238,A -85,B 0,C 180,E1 -10249.849,E2 -10249.849} C_VEL
LIN {X 0,Y 418.239,Z 752.475,A -85,B 0,C 180,E1 -10250.814,E2 -10250.814} C_VEL
LIN {X 0,Y 417.812,Z 759.842,A -85,B 0,C 180,E1 -10252.023,E2 -10252.023} C_VEL
LIN {X 0,Y 417.563,Z 765.601,A -85,B 0,C 180,E1 -10253.234,E2 -10253.234} C_VEL
LIN {X 0,Y 417.429,Z 769.353,A -85,B 0,C 180,E1 -10254.202,E2 -10254.202} C_VEL
LIN {X 0,Y 417.141,Z 773.616,A -85,B 0,C 180,E1 -10255.652,E2 -10255.652} C_VEL
LIN {X 0,Y 417.094,Z 776.569,A -85,B 0,C 180,E1 -10257.103,E2 -10257.103} C_VEL
LIN {X 0,Y 417.062,Z 777.822,A -85,B 0,C 180,E1 -10258.069,E2 -10258.069} C_VEL
LIN {X 0,Y 416.992,Z 778.559,A -85,B 0,C 180,E1 -10259.034,E2 -10259.034} C_VEL
LIN {X 0,Y 416.982,Z 778.786,A -85,B 0,C 180,E1 -10260,E2 -10260} C_VEL
LIN {X 0,Y 416.993,Z 778.443,A -85,B 0,C 180,E1 -10260.966,E2 -10260.966} C_VEL
LIN {X 0,Y 417.06,Z 777.515,A -85,B 0,C 180,E1 -10261.931,E2 -10261.931} C_VEL
LIN {X 0,Y 417.058,Z 775.199,A -85,B 0,C 180,E1 -10263.381,E2 -10263.381} C_VEL
LIN {X 0,Y 417.202,Z 771.462,A -85,B 0,C 180,E1 -10264.832,E2 -10264.832} C_VEL
LIN {X 0,Y 417.351,Z 766.495,A -85,B 0,C 180,E1 -10266.235,E2 -10266.235} C_VEL
LIN {X 0,Y 417.585,Z 760.737,A -85,B 0,C 180,E1 -10267.495,E2 -10267.495} C_VEL
LIN {X 0,Y 417.893,Z 753.634,A -85,B 0,C 180,E1 -10268.706,E2 -10268.706} C_VEL
LIN {X 0,Y 418.242,Z 746.581,A -85,B 0,C 180,E1 -10269.674,E2 -10269.674} C_VEL
LIN {X 0,Y 418.632,Z 739.112,A -85,B 0,C 180,E1 -10270.52,E2 -10270.52} C_VEL
LIN {X 0,Y 418.926,Z 731.338,A -85,B 0,C 180,E1 -10271.246,E2 -10271.246} C_VEL
LIN {X 0,Y 419.342,Z 721.684,A -85,B 0,C 180,E1 -10271.97,E2 -10271.97} C_VEL
LIN {X 0,Y 419.735,Z 709.591,A -85,B 0,C 180,E1 -10272.634,E2 -10272.634} C_VEL
LIN {X 0,Y 419.893,Z 700.05,A -85,B 0,C 180,E1 -10272.998,E2 -10272.998} C_VEL
LIN {X 0,Y 420.207,Z 689.252,A -85,B 0,C 180,E1 -10273.265,E2 -10273.265} C_VEL
LIN {X 0,Y 420.856,Z 632.492,A -85,B 0,C 180,E1 -10274.404,E2 -10274.404} C_VEL
LIN {X 0,Y 419.074,Z 617.111,A -85,B 0,C 180,E1 -10274.787,E2 -10274.787} C_VEL
LIN {X 0,Y 419.103,Z 614.989,A -85,B 0,C 180,E1 -10275.066,E2 -10275.066} C_VEL
LIN {X 0,Y 419.7,Z 598.289,A -85,B 0,C 180,E1 -10277.794,E2 -10277.794} C_VEL
LIN {X 0,Y 420.538,Z 578.659,A -85,B 0,C 180,E1 -10281.006,E2 -10281.006} C_VEL
LIN {X 0,Y 421.422,Z 558.124,A -85,B 0,C 180,E1 -10284.378,E2 -10284.378} C_VEL
LIN {X 0,Y 421.673,Z 549.279,A -85,B 0,C 180,E1 -10285.839,E2 -10285.839} C_VEL
LIN {X 0,Y 418.958,Z 535.455,A -85,B 0,C 180,E1 -10288.287,E2 -10288.287} C_VEL
LIN {X 0,Y 418.323,Z 532.461,A -85,B 0,C 180,E1 -10288.882,E2 -10288.882} C_VEL
LIN {X 0,Y 418.249,Z 532.385,A -85,B 0,C 180,E1 -10292.528,E2 -10292.528} C_VEL
LIN {X 0,Y 418.263,Z 532.383,A -85,B 0,C 180,E1 -10294.841,E2 -10294.841} C_VEL
LIN {X 0,Y 418.263,Z 532.38,A -85,B 0,C 180,E1 -10298.441,E2 -10298.441} C_VEL
LIN {X 0,Y 418.224,Z 532.368,A -85,B 0,C 180,E1 -10300.948,E2 -10300.948} C_VEL
LIN {X 0,Y 418.212,Z 532.37,A -85,B 0,C 180,E1 -10303.729,E2 -10303.729} C_VEL
LIN {X 0,Y 418.212,Z 532.388,A -85,B 0,C 180,E1 -10306.448,E2 -10306.448} C_VEL
LIN {X 0,Y 418.227,Z 532.373,A -85,B 0,C 180,E1 -10309.13,E2 -10309.13} C_VEL
LIN {X 0,Y 418.229,Z 532.383,A -85,B 0,C 180,E1 -10312.167,E2 -10312.167} C_VEL
LIN {X 0,Y 418.268,Z 532.378,A -85,B 0,C 180,E1 -10315.42,E2 -10315.42} C_VEL
LIN {X 0,Y 418.215,Z 532.388,A -85,B 0,C 180,E1 -10318.604,E2 -10318.604} C_VEL
LIN {X 0,Y 418.296,Z 532.38,A -85,B 0,C 180,E1 -10321.936,E2 -10321.936} C_VEL
LIN {X 0,Y 418.294,Z 532.373,A -85,B 0,C 180,E1 -10325.162,E2 -10325.162} C_VEL
LIN {X 0,Y 418.328,Z 532.587,A -85,B 0,C 180,E1 -10326.549,E2 -10326.549} C_VEL
LIN {X 0,Y 420.257,Z 542.777,A -85,B 0,C 180,E1 -10329.183,E2 -10329.183} C_VEL
LIN {X 0,Y 420.003,Z 550.129,A -85,B 0,C 180,E1 -10330.911,E2 -10330.911} C_VEL
LIN {X 0,Y 420.101,Z 551.332,A -85,B 0,C 180,E1 -10331.025,E2 -10331.025} C_VEL
LIN {X 0,Y 423.997,Z 570.761,A -85,B 0,C 180,E1 -10331.561,E2 -10331.561} C_VEL
LIN {X 0,Y 423.243,Z 645.385,A -85,B 0,C 180,E1 -10332.831,E2 -10332.831} C_VEL
LIN {X 0,Y 422.492,Z 651.228,A -85,B 0,C 180,E1 -10332.901,E2 -10332.901} C_VEL
LIN {X 0,Y 419.54,Z 660.685,A -85,B 0,C 180,E1 -10332.997,E2 -10332.997} C_VEL
LIN {X 0,Y 416.535,Z 670.005,A -85,B 0,C 180,E1 -10333.187,E2 -10333.187} C_VEL
LIN {X 0,Y 415.67,Z 675.624,A -85,B 0,C 180,E1 -10333.402,E2 -10333.402} C_VEL
LIN {X 0,Y 415.084,Z 687.256,A -85,B 0,C 180,E1 -10334.029,E2 -10334.029} C_VEL
LIN {X 0,Y 414.341,Z 699.254,A -85,B 0,C 180,E1 -10334.882,E2 -10334.882} C_VEL
LIN {X 0,Y 413.641,Z 710.535,A -85,B 0,C 180,E1 -10335.927,E2 -10335.927} C_VEL
LIN {X 0,Y 412.956,Z 719.659,A -85,B 0,C 180,E1 -10336.967,E2 -10336.967} C_VEL
LIN {X 0,Y 412.142,Z 728.505,A -85,B 0,C 180,E1 -10338.192,E2 -10338.192} C_VEL
LIN {X 0,Y 411.489,Z 737.131,A -85,B 0,C 180,E1 -10339.668,E2 -10339.668} C_VEL
LIN {X 0,Y 410.935,Z 744.006,A -85,B 0,C 180,E1 -10341.145,E2 -10341.145} C_VEL
LIN {X 0,Y 410.519,Z 749.512,A -85,B 0,C 180,E1 -10342.622,E2 -10342.622} C_VEL
LIN {X 0,Y 410.345,Z 753.828,A -85,B 0,C 180,E1 -10344.101,E2 -10344.101} C_VEL
LIN {X 0,Y 410.165,Z 756.112,A -85,B 0,C 180,E1 -10345.084,E2 -10345.084} C_VEL
LIN {X 0,Y 410.058,Z 757.971,A -85,B 0,C 180,E1 -10346.068,E2 -10346.068} C_VEL
LIN {X 0,Y 410.06,Z 759.371,A -85,B 0,C 180,E1 -10347.052,E2 -10347.052} C_VEL
LIN {X 0,Y 410.013,Z 760.368,A -85,B 0,C 180,E1 -10348.035,E2 -10348.035} C_VEL
LIN {X 0,Y 409.927,Z 761.219,A -85,B 0,C 180,E1 -10349.999,E2 -10349.999} C_VEL
LIN {X 0,Y 409.939,Z 761.032,A -85,B 0,C 180,E1 -10350.981,E2 -10350.981} C_VEL
LIN {X 0,Y 410.012,Z 760.448,A -85,B 0,C 180,E1 -10351.964,E2 -10351.964} C_VEL
LIN {X 0,Y 410.056,Z 759.483,A -85,B 0,C 180,E1 -10352.946,E2 -10352.946} C_VEL
LIN {X 0,Y 410.046,Z 758.131,A -85,B 0,C 180,E1 -10353.93,E2 -10353.93} C_VEL
LIN {X 0,Y 410.267,Z 755.263,A -85,B 0,C 180,E1 -10355.405,E2 -10355.405} C_VEL
LIN {X 0,Y 410.462,Z 751.377,A -85,B 0,C 180,E1 -10356.883,E2 -10356.883} C_VEL
LIN {X 0,Y 410.756,Z 746.368,A -85,B 0,C 180,E1 -10358.362,E2 -10358.362} C_VEL
LIN {X 0,Y 411.302,Z 740.057,A -85,B 0,C 180,E1 -10359.838,E2 -10359.838} C_VEL
LIN {X 0,Y 411.931,Z 732.156,A -85,B 0,C 180,E1 -10361.314,E2 -10361.314} C_VEL
LIN {X 0,Y 412.539,Z 724.104,A -85,B 0,C 180,E1 -10362.544,E2 -10362.544} C_VEL
LIN {X 0,Y 413.399,Z 714.269,A -85,B 0,C 180,E1 -10363.768,E2 -10363.768} C_VEL
LIN {X 0,Y 414.058,Z 703.22,A -85,B 0,C 180,E1 -10364.875,E2 -10364.875} C_VEL
LIN {X 0,Y 414.772,Z 692.375,A -85,B 0,C 180,E1 -10365.729,E2 -10365.729} C_VEL
LIN {X 0,Y 415.487,Z 680.386,A -85,B 0,C 180,E1 -10366.458,E2 -10366.458} C_VEL
LIN {X 0,Y 415.941,Z 668.116,A -85,B 0,C 180,E1 -10367.008,E2 -10367.008} C_VEL
LIN {X 0,Y 416.379,Z 655.49,A -85,B 0,C 180,E1 -10367.369,E2 -10367.369} C_VEL
LIN {X 0,Y 417.203,Z 571.255,A -85,B 0,C 180,E1 -10368.843,E2 -10368.843} C_VEL
LIN {X 0,Y 413.18,Z 551.195,A -85,B 0,C 180,E1 -10369.416,E2 -10369.416} C_VEL
LIN {X 0,Y 413.119,Z 550.416,A -85,B 0,C 180,E1 -10369.502,E2 -10369.502} C_VEL
LIN {X 0,Y 413.306,Z 544.437,A -85,B 0,C 180,E1 -10370.921,E2 -10370.921} C_VEL
LIN {X 0,Y 411.382,Z 533.886,A -85,B 0,C 180,E1 -10373.669,E2 -10373.669} C_VEL
LIN {X 0,Y 411.248,Z 533.269,A -85,B 0,C 180,E1 -10373.945,E2 -10373.945} C_VEL
LIN {X 0,Y 411.258,Z 533.26,A -85,B 0,C 180,E1 -10377.477,E2 -10377.477} C_VEL
LIN {X 0,Y 411.188,Z 533.262,A -85,B 0,C 180,E1 -10380.846,E2 -10380.846} C_VEL
LIN {X 0,Y 411.204,Z 533.263,A -85,B 0,C 180,E1 -10384.332,E2 -10384.332} C_VEL
LIN {X 0,Y 411.198,Z 533.263,A -85,B 0,C 180,E1 -10387.972,E2 -10387.972} C_VEL
LIN {X 0,Y 411.19,Z 533.263,A -85,B 0,C 180,E1 -10391.232,E2 -10391.232} C_VEL
LIN {X 0,Y 411.175,Z 533.256,A -85,B 0,C 180,E1 -10394.489,E2 -10394.489} C_VEL
LIN {X 0,Y 411.194,Z 533.262,A -85,B 0,C 180,E1 -10398.196,E2 -10398.196} C_VEL
LIN {X 0,Y 411.227,Z 533.248,A -85,B 0,C 180,E1 -10400.777,E2 -10400.777} C_VEL
LIN {X 0,Y 411.196,Z 533.261,A -85,B 0,C 180,E1 -10404.471,E2 -10404.471} C_VEL
LIN {X 0,Y 411.162,Z 533.265,A -85,B 0,C 180,E1 -10408.002,E2 -10408.002} C_VEL
LIN {X 0,Y 411.218,Z 533.26,A -85,B 0,C 180,E1 -10411.41,E2 -10411.41} C_VEL
LIN {X 0,Y 411.23,Z 533.257,A -85,B 0,C 180,E1 -10414.706,E2 -10414.706} C_VEL
LIN {X 0,Y 411.198,Z 533.258,A -85,B 0,C 180,E1 -10417.913,E2 -10417.913} C_VEL
LIN {X 0,Y 411.218,Z 533.26,A -85,B 0,C 180,E1 -10421.051,E2 -10421.051} C_VEL
LIN {X 0,Y 411.247,Z 533.25,A -85,B 0,C 180,E1 -10424.131,E2 -10424.131} C_VEL
LIN {X 0,Y 411.295,Z 533.251,A -85,B 0,C 180,E1 -10427.165,E2 -10427.165} C_VEL
LIN {X 0,Y 411.286,Z 533.242,A -85,B 0,C 180,E1 -10430.161,E2 -10430.161} C_VEL
LIN {X 0,Y 411.453,Z 533.231,A -85,B 0,C 180,E1 -10433.133,E2 -10433.133} C_VEL
LIN {X 0,Y 411.305,Z 533.249,A -85,B 0,C 180,E1 -10435.099,E2 -10435.099} C_VEL
LIN {X 0,Y 411.506,Z 533.222,A -85,B 0,C 180,E1 -10438.042,E2 -10438.042} C_VEL
LIN {X 0,Y 411.636,Z 533.209,A -85,B 0,C 180,E1 -10440,E2 -10440} C_VEL
LIN {X 0,Y 411.46,Z 533.224,A -85,B 0,C 180,E1 -10442.937,E2 -10442.937} C_VEL
LIN {X 0,Y 411.481,Z 533.229,A -85,B 0,C 180,E1 -10445.882,E2 -10445.882} C_VEL
LIN {X 0,Y 411.474,Z 533.228,A -85,B 0,C 180,E1 -10447.853,E2 -10447.853} C_VEL
LIN {X 0,Y 411.291,Z 533.253,A -85,B 0,C 180,E1 -10451.833,E2 -10451.833} C_VEL
LIN {X 0,Y 411.255,Z 533.252,A -85,B 0,C 180,E1 -10454.853,E2 -10454.853} C_VEL
LIN {X 0,Y 411.245,Z 533.259,A -85,B 0,C 180,E1 -10457.915,E2 -10457.915} C_VEL
LIN {X 0,Y 411.195,Z 533.26,A -85,B 0,C 180,E1 -10461.034,E2 -10461.034} C_VEL
LIN {X 0,Y 411.22,Z 533.26,A -85,B 0,C 180,E1 -10464.216,E2 -10464.216} C_VEL
LIN {X 0,Y 411.252,Z 533.254,A -85,B 0,C 180,E1 -10467.478,E2 -10467.478} C_VEL
LIN {X 0,Y 411.184,Z 533.26,A -85,B 0,C 180,E1 -10470.848,E2 -10470.848} C_VEL
LIN {X 0,Y 411.2,Z 533.258,A -85,B 0,C 180,E1 -10474.334,E2 -10474.334} C_VEL
LIN {X 0,Y 411.196,Z 533.26,A -85,B 0,C 180,E1 -10477.974,E2 -10477.974} C_VEL
LIN {X 0,Y 411.178,Z 533.263,A -85,B 0,C 180,E1 -10480.505,E2 -10480.505} C_VEL
LIN {X 0,Y 411.169,Z 533.257,A -85,B 0,C 180,E1 -10483.134,E2 -10483.134} C_VEL
LIN {X 0,Y 411.223,Z 533.258,A -85,B 0,C 180,E1 -10485.873,E2 -10485.873} C_VEL
LIN {X 0,Y 411.206,Z 533.261,A -85,B 0,C 180,E1 -10488.765,E2 -10488.765} C_VEL
LIN {X 0,Y 411.201,Z 533.243,A -85,B 0,C 180,E1 -10492.028,E2 -10492.028} C_VEL
LIN {X 0,Y 411.203,Z 533.26,A -85,B 0,C 180,E1 -10495.668,E2 -10495.668} C_VEL
LIN {X 0,Y 411.187,Z 533.212,A -85,B 0,C 180,E1 -10499.153,E2 -10499.153} C_VEL
LIN {X 0,Y 411.306,Z 533.44,A -85,B 0,C 180,E1 -10502.251,E2 -10502.251} C_VEL
LIN {X 0,Y 413.867,Z 546.036,A -85,B 0,C 180,E1 -10505.148,E2 -10505.148} C_VEL
LIN {X 0,Y 414.399,Z 549.84,A -85,B 0,C 180,E1 -10505.983,E2 -10505.983} C_VEL
LIN {X 0,Y 413.263,Z 565.894,A -85,B 0,C 180,E1 -10509.283,E2 -10509.283} C_VEL
LIN {X 0,Y 412.873,Z 572.513,A -85,B 0,C 180,E1 -10510.583,E2 -10510.583} C_VEL
LIN {X 0,Y 417.011,Z 597.954,A -85,B 0,C 180,E1 -10511.264,E2 -10511.264} C_VEL
LIN {X 0,Y 416.138,Z 680.568,A -85,B 0,C 180,E1 -10512.715,E2 -10512.715} C_VEL
LIN {X 0,Y 415.555,Z 693.796,A -85,B 0,C 180,E1 -10513.134,E2 -10513.134} C_VEL
LIN {X 0,Y 414.914,Z 707.065,A -85,B 0,C 180,E1 -10513.772,E2 -10513.772} C_VEL
LIN {X 0,Y 414.163,Z 718.211,A -85,B 0,C 180,E1 -10514.499,E2 -10514.499} C_VEL
LIN {X 0,Y 413.341,Z 729.885,A -85,B 0,C 180,E1 -10515.485,E2 -10515.485} C_VEL
LIN {X 0,Y 412.591,Z 740.241,A -85,B 0,C 180,E1 -10516.581,E2 -10516.581} C_VEL
LIN {X 0,Y 411.954,Z 748.78,A -85,B 0,C 180,E1 -10517.688,E2 -10517.688} C_VEL
LIN {X 0,Y 411.322,Z 756.657,A -85,B 0,C 180,E1 -10518.918,E2 -10518.918} C_VEL
LIN {X 0,Y 410.762,Z 764.353,A -85,B 0,C 180,E1 -10520.398,E2 -10520.398} C_VEL
LIN {X 0,Y 410.341,Z 771.45,A -85,B 0,C 180,E1 -10522.126,E2 -10522.126} C_VEL
LIN {X 0,Y 410.043,Z 776.658,A -85,B 0,C 180,E1 -10523.775,E2 -10523.775} C_VEL
LIN {X 0,Y 410.025,Z 779.786,A -85,B 0,C 180,E1 -10525.084,E2 -10525.084} C_VEL
LIN {X 0,Y 409.935,Z 781.648,A -85,B 0,C 180,E1 -10526.069,E2 -10526.069} C_VEL
LIN {X 0,Y 409.966,Z 784.04,A -85,B 0,C 180,E1 -10528.036,E2 -10528.036} C_VEL
LIN {X 0,Y 409.926,Z 785.117,A -85,B 0,C 180,E1 -10530.001,E2 -10530.001} C_VEL
LIN {X 0,Y 409.935,Z 784.924,A -85,B 0,C 180,E1 -10530.983,E2 -10530.983} C_VEL
LIN {X 0,Y 409.967,Z 784.221,A -85,B 0,C 180,E1 -10531.966,E2 -10531.966} C_VEL
LIN {X 0,Y 409.935,Z 781.635,A -85,B 0,C 180,E1 -10533.933,E2 -10533.933} C_VEL
LIN {X 0,Y 410.028,Z 778.698,A -85,B 0,C 180,E1 -10535.41,E2 -10535.41} C_VEL
LIN {X 0,Y 410.169,Z 774.723,A -85,B 0,C 180,E1 -10536.889,E2 -10536.889} C_VEL
LIN {X 0,Y 410.493,Z 768.605,A -85,B 0,C 180,E1 -10538.617,E2 -10538.617} C_VEL
LIN {X 0,Y 410.939,Z 761.924,A -85,B 0,C 180,E1 -10540.097,E2 -10540.097} C_VEL
LIN {X 0,Y 411.543,Z 753.637,A -85,B 0,C 180,E1 -10541.576,E2 -10541.576} C_VEL
LIN {X 0,Y 412.253,Z 745.145,A -85,B 0,C 180,E1 -10542.805,E2 -10542.805} C_VEL
LIN {X 0,Y 412.984,Z 734.338,A -85,B 0,C 180,E1 -10544.068,E2 -10544.068} C_VEL
LIN {X 0,Y 413.831,Z 722.835,A -85,B 0,C 180,E1 -10545.137,E2 -10545.137} C_VEL
LIN {X 0,Y 414.652,Z 710.964,A -85,B 0,C 180,E1 -10545.988,E2 -10545.988} C_VEL
LIN {X 0,Y 415.346,Z 698.611,A -85,B 0,C 180,E1 -10546.655,E2 -10546.655} C_VEL
LIN {X 0,Y 415.915,Z 685.912,A -85,B 0,C 180,E1 -10547.137,E2 -10547.137} C_VEL
LIN {X 0,Y 416.286,Z 672.597,A -85,B 0,C 180,E1 -10547.438,E2 -10547.438} C_VEL
LIN {X 0,Y 416.9,Z 597.593,A -85,B 0,C 180,E1 -10548.742,E2 -10548.742} C_VEL
LIN {X 0,Y 412.901,Z 572.922,A -85,B 0,C 180,E1 -10549.385,E2 -10549.385} C_VEL
LIN {X 0,Y 412.873,Z 571.798,A -85,B 0,C 180,E1 -10549.516,E2 -10549.516} C_VEL
LIN {X 0,Y 414.228,Z 553.166,A -85,B 0,C 180,E1 -10553.32,E2 -10553.32} C_VEL
LIN {X 0,Y 414.274,Z 548.527,A -85,B 0,C 180,E1 -10554.293,E2 -10554.293} C_VEL
LIN {X 0,Y 412.095,Z 537.089,A -85,B 0,C 180,E1 -10556.869,E2 -10556.869} C_VEL
LIN {X 0,Y 411.274,Z 533.301,A -85,B 0,C 180,E1 -10557.823,E2 -10557.823} C_VEL
LIN {X 0,Y 411.186,Z 533.266,A -85,B 0,C 180,E1 -10561.284,E2 -10561.284} C_VEL
LIN {X 0,Y 411.21,Z 533.265,A -85,B 0,C 180,E1 -10564.334,E2 -10564.334} C_VEL
LIN {X 0,Y 411.198,Z 533.267,A -85,B 0,C 180,E1 -10567.974,E2 -10567.974} C_VEL
LIN {X 0,Y 411.167,Z 533.268,A -85,B 0,C 180,E1 -10571.229,E2 -10571.229} C_VEL
LIN {X 0,Y 411.179,Z 533.267,A -85,B 0,C 180,E1 -10574.491,E2 -10574.491} C_VEL
LIN {X 0,Y 411.181,Z 533.267,A -85,B 0,C 180,E1 -10578.195,E2 -10578.195} C_VEL
LIN {X 0,Y 411.227,Z 533.26,A -85,B 0,C 180,E1 -10580.777,E2 -10580.777} C_VEL
LIN {X 0,Y 411.203,Z 533.266,A -85,B 0,C 180,E1 -10584.472,E2 -10584.472} C_VEL
LIN {X 0,Y 411.211,Z 533.264,A -85,B 0,C 180,E1 -10586.874,E2 -10586.874} C_VEL
LIN {X 0,Y 411.238,Z 533.425,A -85,B 0,C 180,E1 -10590.114,E2 -10590.114} C_VEL
LIN {X 0,Y 413.88,Z 542.837,A -85,B 0,C 180,E1 -10592.007,E2 -10592.007} C_VEL
LIN {X 0,Y 415.655,Z 551.696,A -85,B 0,C 180,E1 -10593.656,E2 -10593.656} C_VEL
LIN {X 0,Y 415.53,Z 559.709,A -85,B 0,C 180,E1 -10594.986,E2 -10594.986} C_VEL
LIN {X 0,Y 414.449,Z 580.402,A -85,B 0,C 180,E1 -10598.383,E2 -10598.383} C_VEL
LIN {X 0,Y 413.417,Z 602.087,A -85,B 0,C 180,E1 -10601.926,E2 -10601.926} C_VEL
LIN {X 0,Y 412.825,Z 617.138,A -85,B 0,C 180,E1 -10604.352,E2 -10604.352} C_VEL
LIN {X 0,Y 414.791,Z 630.335,A -85,B 0,C 180,E1 -10604.792,E2 -10604.792} C_VEL
LIN {X 0,Y 415.102,Z 636.717,A -85,B 0,C 180,E1 -10604.961,E2 -10604.961} C_VEL
LIN {X 0,Y 413.885,Z 698.187,A -85,B 0,C 180,E1 -10606.341,E2 -10606.341} C_VEL
LIN {X 0,Y 413.525,Z 707.385,A -85,B 0,C 180,E1 -10606.674,E2 -10606.674} C_VEL
LIN {X 0,Y 413.212,Z 716.993,A -85,B 0,C 180,E1 -10607.163,E2 -10607.163} C_VEL
LIN {X 0,Y 412.756,Z 727.047,A -85,B 0,C 180,E1 -10607.836,E2 -10607.836} C_VEL
LIN {X 0,Y 412.233,Z 736.815,A -85,B 0,C 180,E1 -10608.693,E2 -10608.693} C_VEL
LIN {X 0,Y 411.808,Z 743.656,A -85,B 0,C 180,E1 -10609.429,E2 -10609.429} C_VEL
LIN {X 0,Y 411.374,Z 751.163,A -85,B 0,C 180,E1 -10610.412,E2 -10610.412} C_VEL
LIN {X 0,Y 410.952,Z 757.366,A -85,B 0,C 180,E1 -10611.394,E2 -10611.394} C_VEL
LIN {X 0,Y 410.675,Z 762.519,A -85,B 0,C 180,E1 -10612.379,E2 -10612.379} C_VEL
LIN {X 0,Y 410.457,Z 767.672,A -85,B 0,C 180,E1 -10613.587,E2 -10613.587} C_VEL
LIN {X 0,Y 410.157,Z 772.607,A -85,B 0,C 180,E1 -10615.085,E2 -10615.085} C_VEL
LIN {X 0,Y 410.02,Z 774.959,A -85,B 0,C 180,E1 -10616.069,E2 -10616.069} C_VEL
LIN {X 0,Y 409.997,Z 776.711,A -85,B 0,C 180,E1 -10617.052,E2 -10617.052} C_VEL
LIN {X 0,Y 409.975,Z 777.93,A -85,B 0,C 180,E1 -10618.035,E2 -10618.035} C_VEL
LIN {X 0,Y 409.919,Z 778.633,A -85,B 0,C 180,E1 -10619.018,E2 -10619.018} C_VEL
LIN {X 0,Y 409.905,Z 778.827,A -85,B 0,C 180,E1 -10620,E2 -10620} C_VEL
LIN {X 0,Y 409.919,Z 778.471,A -85,B 0,C 180,E1 -10620.982,E2 -10620.982} C_VEL
LIN {X 0,Y 409.972,Z 777.516,A -85,B 0,C 180,E1 -10621.965,E2 -10621.965} C_VEL
LIN {X 0,Y 409.964,Z 775.133,A -85,B 0,C 180,E1 -10623.44,E2 -10623.44} C_VEL
LIN {X 0,Y 410.117,Z 771.326,A -85,B 0,C 180,E1 -10624.915,E2 -10624.915} C_VEL
LIN {X 0,Y 410.246,Z 766.901,A -85,B 0,C 180,E1 -10626.189,E2 -10626.189} C_VEL
LIN {X 0,Y 410.492,Z 761.65,A -85,B 0,C 180,E1 -10627.378,E2 -10627.378} C_VEL
LIN {X 0,Y 410.77,Z 754.86,A -85,B 0,C 180,E1 -10628.61,E2 -10628.61} C_VEL
LIN {X 0,Y 411.217,Z 746.071,A -85,B 0,C 180,E1 -10629.841,E2 -10629.841} C_VEL
LIN {X 0,Y 411.628,Z 738.486,A -85,B 0,C 180,E1 -10630.701,E2 -10630.701} C_VEL
LIN {X 0,Y 412.025,Z 729.149,A -85,B 0,C 180,E1 -10631.562,E2 -10631.562} C_VEL
LIN {X 0,Y 412.491,Z 717.641,A -85,B 0,C 180,E1 -10632.359,E2 -10632.359} C_VEL
LIN {X 0,Y 412.732,Z 708.028,A -85,B 0,C 180,E1 -10632.852,E2 -10632.852} C_VEL
LIN {X 0,Y 413.032,Z 697.921,A -85,B 0,C 180,E1 -10633.218,E2 -10633.218} C_VEL
LIN {X 0,Y 413.537,Z 665.501,A -85,B 0,C 180,E1 -10633.905,E2 -10633.905} C_VEL
LIN {X 0,Y 413.79,Z 632.242,A -85,B 0,C 180,E1 -10634.603,E2 -10634.603} C_VEL
LIN {X 0,Y 412.056,Z 616.754,A -85,B 0,C 180,E1 -10635.013,E2 -10635.013} C_VEL
LIN {X 0,Y 412.694,Z 599.404,A -85,B 0,C 180,E1 -10637.85,E2 -10637.85} C_VEL
LIN {X 0,Y 413.634,Z 577.757,A -85,B 0,C 180,E1 -10641.426,E2 -10641.426} C_VEL
LIN {X 0,Y 414.485,Z 558.948,A -85,B 0,C 180,E1 -10644.546,E2 -10644.546} C_VEL
LIN {X 0,Y 414.751,Z 550.802,A -85,B 0,C 180,E1 -10645.905,E2 -10645.905} C_VEL
LIN {X 0,Y 412.156,Z 537.469,A -85,B 0,C 180,E1 -10648.29,E2 -10648.29} C_VEL
LIN {X 0,Y 411.253,Z 533.374,A -85,B 0,C 180,E1 -10649.073,E2 -10649.073} C_VEL
LIN {X 0,Y 411.17,Z 533.271,A -85,B 0,C 180,E1 -10651.997,E2 -10651.997} C_VEL
LIN {X 0,Y 411.215,Z 533.261,A -85,B 0,C 180,E1 -10654.878,E2 -10654.878} C_VEL
LIN {X 0,Y 411.214,Z 533.259,A -85,B 0,C 180,E1 -10658.169,E2 -10658.169} C_VEL
LIN {X 0,Y 411.164,Z 533.241,A -85,B 0,C 180,E1 -10661.228,E2 -10661.228} C_VEL
LIN {X 0,Y 411.179,Z 533.255,A -85,B 0,C 180,E1 -10664.49,E2 -10664.49} C_VEL
LIN {X 0,Y 411.181,Z 533.259,A -85,B 0,C 180,E1 -10668.194,E2 -10668.194} C_VEL
LIN {X 0,Y 411.212,Z 533.238,A -85,B 0,C 180,E1 -10670.774,E2 -10670.774} C_VEL
LIN {X 0,Y 411.201,Z 533.262,A -85,B 0,C 180,E1 -10674.471,E2 -10674.471} C_VEL
LIN {X 0,Y 411.211,Z 533.262,A -85,B 0,C 180,E1 -10676.873,E2 -10676.873} C_VEL
LIN {X 0,Y 411.237,Z 533.262,A -85,B 0,C 180,E1 -10680.644,E2 -10680.644} C_VEL
LIN {X 0,Y 411.242,Z 533.258,A -85,B 0,C 180,E1 -10683.619,E2 -10683.619} C_VEL
LIN {X 0,Y 411.279,Z 533.361,A -85,B 0,C 180,E1 -10686.256,E2 -10686.256} C_VEL
LIN {X 0,Y 413.364,Z 544.707,A -85,B 0,C 180,E1 -10689.246,E2 -10689.246} C_VEL
LIN {X 0,Y 413.126,Z 550.759,A -85,B 0,C 180,E1 -10690.649,E2 -10690.649} C_VEL
LIN {X 0,Y 414.571,Z 557.785,A -85,B 0,C 180,E1 -10690.887,E2 -10690.887} C_VEL
LIN {X 0,Y 417.283,Z 572.094,A -85,B 0,C 180,E1 -10691.273,E2 -10691.273} C_VEL
LIN {X 0,Y 416.253,Z 656.858,A -85,B 0,C 180,E1 -10692.75,E2 -10692.75} C_VEL
LIN {X 0,Y 415.874,Z 670.367,A -85,B 0,C 180,E1 -10693.177,E2 -10693.177} C_VEL
LIN {X 0,Y 415.67,Z 675.624,A -85,B 0,C 180,E1 -10693.402,E2 -10693.402} C_VEL
LIN {X 0,Y 414.729,Z 681.269,A -85,B 0,C 180,E1 -10693.652,E2 -10693.652} C_VEL
LIN {X 0,Y 411.47,Z 690.213,A -85,B 0,C 180,E1 -10694.074,E2 -10694.074} C_VEL
LIN {X 0,Y 408.177,Z 698.717,A -85,B 0,C 180,E1 -10694.589,E2 -10694.589} C_VEL
LIN {X 0,Y 407.208,Z 703.671,A -85,B 0,C 180,E1 -10694.988,E2 -10694.988} C_VEL
LIN {X 0,Y 406.481,Z 714.719,A -85,B 0,C 180,E1 -10696.119,E2 -10696.119} C_VEL
LIN {X 0,Y 405.664,Z 723.623,A -85,B 0,C 180,E1 -10697.238,E2 -10697.238} C_VEL
LIN {X 0,Y 405.015,Z 731.789,A -85,B 0,C 180,E1 -10698.488,E2 -10698.488} C_VEL
LIN {X 0,Y 404.335,Z 739.788,A -85,B 0,C 180,E1 -10699.989,E2 -10699.989} C_VEL
LIN {X 0,Y 403.721,Z 746.213,A -85,B 0,C 180,E1 -10701.49,E2 -10701.49} C_VEL
LIN {X 0,Y 403.347,Z 752.19,A -85,B 0,C 180,E1 -10703.307,E2 -10703.307} C_VEL
LIN {X 0,Y 403.11,Z 756.317,A -85,B 0,C 180,E1 -10704.998,E2 -10704.998} C_VEL
LIN {X 0,Y 402.975,Z 758.177,A -85,B 0,C 180,E1 -10705.999,E2 -10705.999} C_VEL
LIN {X 0,Y 402.964,Z 759.576,A -85,B 0,C 180,E1 -10707,E2 -10707} C_VEL
LIN {X 0,Y 402.945,Z 760.573,A -85,B 0,C 180,E1 -10708,E2 -10708} C_VEL
LIN {X 0,Y 402.851,Z 761.423,A -85,B 0,C 180,E1 -10709.999,E2 -10709.999} C_VEL
LIN {X 0,Y 402.867,Z 761.236,A -85,B 0,C 180,E1 -10710.999,E2 -10710.999} C_VEL
LIN {X 0,Y 402.945,Z 760.651,A -85,B 0,C 180,E1 -10711.998,E2 -10711.998} C_VEL
LIN {X 0,Y 402.959,Z 759.688,A -85,B 0,C 180,E1 -10712.998,E2 -10712.998} C_VEL
LIN {X 0,Y 402.964,Z 758.335,A -85,B 0,C 180,E1 -10713.999,E2 -10713.999} C_VEL
LIN {X 0,Y 403.215,Z 755.466,A -85,B 0,C 180,E1 -10715.5,E2 -10715.5} C_VEL
LIN {X 0,Y 403.403,Z 751.58,A -85,B 0,C 180,E1 -10717.004,E2 -10717.004} C_VEL
LIN {X 0,Y 403.716,Z 746.571,A -85,B 0,C 180,E1 -10718.508,E2 -10718.508} C_VEL
LIN {X 0,Y 404.282,Z 740.261,A -85,B 0,C 180,E1 -10720.01,E2 -10720.01} C_VEL
LIN {X 0,Y 404.96,Z 732.358,A -85,B 0,C 180,E1 -10721.511,E2 -10721.511} C_VEL
LIN {X 0,Y 405.618,Z 724.305,A -85,B 0,C 180,E1 -10722.762,E2 -10722.762} C_VEL
LIN {X 0,Y 406.5,Z 714.47,A -85,B 0,C 180,E1 -10724.006,E2 -10724.006} C_VEL
LIN {X 0,Y 407.209,Z 703.419,A -85,B 0,C 180,E1 -10725.131,E2 -10725.131} C_VEL
LIN {X 0,Y 407.951,Z 692.573,A -85,B 0,C 180,E1 -10725.999,E2 -10725.999} C_VEL
LIN {X 0,Y 408.706,Z 680.582,A -85,B 0,C 180,E1 -10726.739,E2 -10726.739} C_VEL
LIN {X 0,Y 409.178,Z 668.308,A -85,B 0,C 180,E1 -10727.298,E2 -10727.298} C_VEL
LIN {X 0,Y 409.631,Z 655.672,A -85,B 0,C 180,E1 -10727.665,E2 -10727.665} C_VEL
LIN {X 0,Y 410.545,Z 572.454,A -85,B 0,C 180,E1 -10729.141,E2 -10729.141} C_VEL
LIN {X 0,Y 406.256,Z 551.18,A -85,B 0,C 180,E1 -10729.772,E2 -10729.772} C_VEL
LIN {X 0,Y 406.319,Z 548.894,A -85,B 0,C 180,E1 -10730.238,E2 -10730.238} C_VEL
LIN {X 0,Y 406.192,Z 544.632,A -85,B 0,C 180,E1 -10731.305,E2 -10731.305} C_VEL
LIN {X 0,Y 404.227,Z 534.223,A -85,B 0,C 180,E1 -10734.114,E2 -10734.114} C_VEL
LIN {X 0,Y 404.225,Z 534.136,A -85,B 0,C 180,E1 -10737.537,E2 -10737.537} C_VEL
LIN {X 0,Y 404.144,Z 534.137,A -85,B 0,C 180,E1 -10740.284,E2 -10740.284} C_VEL
LIN {X 0,Y 404.143,Z 534.145,A -85,B 0,C 180,E1 -10743.811,E2 -10743.811} C_VEL
LIN {X 0,Y 404.137,Z 534.139,A -85,B 0,C 180,E1 -10746.875,E2 -10746.875} C_VEL
LIN {X 0,Y 404.156,Z 534.134,A -85,B 0,C 180,E1 -10750.081,E2 -10750.081} C_VEL
LIN {X 0,Y 404.153,Z 534.143,A -85,B 0,C 180,E1 -10753.083,E2 -10753.083} C_VEL
LIN {X 0,Y 404.144,Z 534.139,A -85,B 0,C 180,E1 -10755.925,E2 -10755.925} C_VEL
LIN {X 0,Y 404.147,Z 534.14,A -85,B 0,C 180,E1 -10758.638,E2 -10758.638} C_VEL
LIN {X 0,Y 404.157,Z 534.125,A -85,B 0,C 180,E1 -10761.49,E2 -10761.49} C_VEL
LIN {X 0,Y 404.182,Z 534.137,A -85,B 0,C 180,E1 -10764.983,E2 -10764.983} C_VEL
LIN {X 0,Y 404.14,Z 534.138,A -85,B 0,C 180,E1 -10768.553,E2 -10768.553} C_VEL
LIN {X 0,Y 404.192,Z 534.128,A -85,B 0,C 180,E1 -10772,E2 -10772} C_VEL
LIN {X 0,Y 404.171,Z 534.142,A -85,B 0,C 180,E1 -10775.334,E2 -10775.334} C_VEL
LIN {X 0,Y 404.132,Z 534.135,A -85,B 0,C 180,E1 -10778.58,E2 -10778.58} C_VEL
LIN {X 0,Y 404.203,Z 534.133,A -85,B 0,C 180,E1 -10781.761,E2 -10781.761} C_VEL
LIN {X 0,Y 404.199,Z 534.127,A -85,B 0,C 180,E1 -10784.882,E2 -10784.882} C_VEL
LIN {X 0,Y 404.249,Z 534.126,A -85,B 0,C 180,E1 -10787.958,E2 -10787.958} C_VEL
LIN {X 0,Y 404.425,Z 534.105,A -85,B 0,C 180,E1 -10792.099,E2 -10792.099} C_VEL
LIN {X 0,Y 404.417,Z 534.107,A -85,B 0,C 180,E1 -10794.015,E2 -10794.015} C_VEL
LIN {X 0,Y 404.475,Z 534.098,A -85,B 0,C 180,E1 -10798.008,E2 -10798.008} C_VEL
LIN {X 0,Y 404.606,Z 534.085,A -85,B 0,C 180,E1 -10800,E2 -10800} C_VEL
LIN {X 0,Y 404.417,Z 534.102,A -85,B 0,C 180,E1 -10802.988,E2 -10802.988} C_VEL
LIN {X 0,Y 404.427,Z 534.107,A -85,B 0,C 180,E1 -10805.985,E2 -10805.985} C_VEL
LIN {X 0,Y 404.415,Z 534.106,A -85,B 0,C 180,E1 -10807.991,E2 -10807.991} C_VEL
LIN {X 0,Y 404.262,Z 534.127,A -85,B 0,C 180,E1 -10812.041,E2 -10812.041} C_VEL
LIN {X 0,Y 404.2,Z 534.133,A -85,B 0,C 180,E1 -10815.118,E2 -10815.118} C_VEL
LIN {X 0,Y 404.206,Z 534.133,A -85,B 0,C 180,E1 -10818.238,E2 -10818.238} C_VEL
LIN {X 0,Y 404.156,Z 534.138,A -85,B 0,C 180,E1 -10821.418,E2 -10821.418} C_VEL
LIN {X 0,Y 404.17,Z 534.137,A -85,B 0,C 180,E1 -10824.666,E2 -10824.666} C_VEL
LIN {X 0,Y 404.188,Z 534.138,A -85,B 0,C 180,E1 -10828,E2 -10828} C_VEL
LIN {X 0,Y 404.135,Z 534.142,A -85,B 0,C 180,E1 -10831.559,E2 -10831.559} C_VEL
LIN {X 0,Y 404.18,Z 534.133,A -85,B 0,C 180,E1 -10835.017,E2 -10835.017} C_VEL
LIN {X 0,Y 404.154,Z 534.138,A -85,B 0,C 180,E1 -10838.757,E2 -10838.757} C_VEL
LIN {X 0,Y 404.118,Z 534.14,A -85,B 0,C 180,E1 -10841.601,E2 -10841.601} C_VEL
LIN {X 0,Y 404.15,Z 534.14,A -85,B 0,C 180,E1 -10844.524,E2 -10844.524} C_VEL
LIN {X 0,Y 404.203,Z 534.129,A -85,B 0,C 180,E1 -10847.306,E2 -10847.306} C_VEL
LIN {X 0,Y 404.165,Z 534.136,A -85,B 0,C 180,E1 -10849.956,E2 -10849.956} C_VEL
LIN {X 0,Y 404.137,Z 534.129,A -85,B 0,C 180,E1 -10853.125,E2 -10853.125} C_VEL
LIN {X 0,Y 404.142,Z 534.133,A -85,B 0,C 180,E1 -10856.189,E2 -10856.189} C_VEL
LIN {X 0,Y 404.143,Z 534.093,A -85,B 0,C 180,E1 -10859.716,E2 -10859.716} C_VEL
LIN {X 0,Y 404.267,Z 534.351,A -85,B 0,C 180,E1 -10861.972,E2 -10861.972} C_VEL
LIN {X 0,Y 406.854,Z 547.106,A -85,B 0,C 180,E1 -10864.964,E2 -10864.964} C_VEL
LIN {X 0,Y 407.442,Z 552.195,A -85,B 0,C 180,E1 -10866.093,E2 -10866.093} C_VEL
LIN {X 0,Y 406.221,Z 568.069,A -85,B 0,C 180,E1 -10869.411,E2 -10869.411} C_VEL
LIN {X 0,Y 405.96,Z 572.311,A -85,B 0,C 180,E1 -10870.239,E2 -10870.239} C_VEL
LIN {X 0,Y 410.309,Z 599.275,A -85,B 0,C 180,E1 -10870.973,E2 -10870.973} C_VEL
LIN {X 0,Y 409.353,Z 680.375,A -85,B 0,C 180,E1 -10872.42,E2 -10872.42} C_VEL
LIN {X 0,Y 408.785,Z 693.599,A -85,B 0,C 180,E1 -10872.846,E2 -10872.846} C_VEL
LIN {X 0,Y 408.108,Z 706.866,A -85,B 0,C 180,E1 -10873.493,E2 -10873.493} C_VEL
LIN {X 0,Y 407.319,Z 718.01,A -85,B 0,C 180,E1 -10874.232,E2 -10874.232} C_VEL
LIN {X 0,Y 406.436,Z 729.86,A -85,B 0,C 180,E1 -10875.25,E2 -10875.25} C_VEL
LIN {X 0,Y 405.657,Z 740.039,A -85,B 0,C 180,E1 -10876.347,E2 -10876.347} C_VEL
LIN {X 0,Y 405,Z 748.577,A -85,B 0,C 180,E1 -10877.473,E2 -10877.473} C_VEL
LIN {X 0,Y 404.323,Z 756.453,A -85,B 0,C 180,E1 -10878.724,E2 -10878.724} C_VEL
LIN {X 0,Y 403.722,Z 764.149,A -85,B 0,C 180,E1 -10880.229,E2 -10880.229} C_VEL
LIN {X 0,Y 403.287,Z 771.245,A -85,B 0,C 180,E1 -10881.987,E2 -10881.987} C_VEL
LIN {X 0,Y 402.957,Z 776.787,A -85,B 0,C 180,E1 -10883.796,E2 -10883.796} C_VEL
LIN {X 0,Y 402.937,Z 779.582,A -85,B 0,C 180,E1 -10884.998,E2 -10884.998} C_VEL
LIN {X 0,Y 402.855,Z 781.443,A -85,B 0,C 180,E1 -10885.999,E2 -10885.999} C_VEL
LIN {X 0,Y 402.864,Z 783.836,A -85,B 0,C 180,E1 -10888.001,E2 -10888.001} C_VEL
LIN {X 0,Y 402.862,Z 784.634,A -85,B 0,C 180,E1 -10889.001,E2 -10889.001} C_VEL
LIN {X 0,Y 402.851,Z 785.021,A -85,B 0,C 180,E1 -10890.001,E2 -10890.001} C_VEL
LIN {X 0,Y 402.862,Z 784.875,A -85,B 0,C 180,E1 -10891,E2 -10891} C_VEL
LIN {X 0,Y 402.864,Z 784.206,A -85,B 0,C 180,E1 -10892,E2 -10892} C_VEL
LIN {X 0,Y 402.826,Z 783.046,A -85,B 0,C 180,E1 -10893.001,E2 -10893.001} C_VEL
LIN {X 0,Y 402.938,Z 779.565,A -85,B 0,C 180,E1 -10895.004,E2 -10895.004} C_VEL
LIN {X 0,Y 403.006,Z 775.951,A -85,B 0,C 180,E1 -10896.509,E2 -10896.509} C_VEL
LIN {X 0,Y 403.289,Z 771.222,A -85,B 0,C 180,E1 -10898.015,E2 -10898.015} C_VEL
LIN {X 0,Y 403.724,Z 764.117,A -85,B 0,C 180,E1 -10899.773,E2 -10899.773} C_VEL
LIN {X 0,Y 404.325,Z 756.412,A -85,B 0,C 180,E1 -10901.278,E2 -10901.278} C_VEL
LIN {X 0,Y 405.163,Z 746.738,A -85,B 0,C 180,E1 -10902.778,E2 -10902.778} C_VEL
LIN {X 0,Y 405.891,Z 736.758,A -85,B 0,C 180,E1 -10904.03,E2 -10904.03} C_VEL
LIN {X 0,Y 406.725,Z 725.485,A -85,B 0,C 180,E1 -10905.151,E2 -10905.151} C_VEL
LIN {X 0,Y 407.532,Z 714.448,A -85,B 0,C 180,E1 -10906.018,E2 -10906.018} C_VEL
LIN {X 0,Y 408.344,Z 702.222,A -85,B 0,C 180,E1 -10906.756,E2 -10906.756} C_VEL
LIN {X 0,Y 408.977,Z 689.364,A -85,B 0,C 180,E1 -10907.308,E2 -10907.308} C_VEL
LIN {X 0,Y 409.474,Z 675.701,A -85,B 0,C 180,E1 -10907.673,E2 -10907.673} C_VEL
LIN {X 0,Y 410.201,Z 598.614,A -85,B 0,C 180,E1 -10909.037,E2 -10909.037} C_VEL
LIN {X 0,Y 405.999,Z 572.702,A -85,B 0,C 180,E1 -10909.728,E2 -10909.728} C_VEL
LIN {X 0,Y 406.01,Z 570.912,A -85,B 0,C 180,E1 -10909.991,E2 -10909.991} C_VEL
LIN {X 0,Y 407.4,Z 552.862,A -85,B 0,C 180,E1 -10913.758,E2 -10913.758} C_VEL
LIN {X 0,Y 407.283,Z 549.594,A -85,B 0,C 180,E1 -10914.466,E2 -10914.466} C_VEL
LIN {X 0,Y 404.985,Z 537.634,A -85,B 0,C 180,E1 -10917.216,E2 -10917.216} C_VEL
LIN {X 0,Y 404.238,Z 534.193,A -85,B 0,C 180,E1 -10918.103,E2 -10918.103} C_VEL
LIN {X 0,Y 404.143,Z 534.143,A -85,B 0,C 180,E1 -10921.558,E2 -10921.558} C_VEL
LIN {X 0,Y 404.188,Z 534.135,A -85,B 0,C 180,E1 -10925.016,E2 -10925.016} C_VEL
LIN {X 0,Y 404.158,Z 534.14,A -85,B 0,C 180,E1 -10928.757,E2 -10928.757} C_VEL
LIN {X 0,Y 404.126,Z 534.146,A -85,B 0,C 180,E1 -10931.6,E2 -10931.6} C_VEL
LIN {X 0,Y 404.149,Z 534.142,A -85,B 0,C 180,E1 -10934.522,E2 -10934.522} C_VEL
LIN {X 0,Y 404.14,Z 534.144,A -85,B 0,C 180,E1 -10937.296,E2 -10937.296} C_VEL
LIN {X 0,Y 404.172,Z 534.14,A -85,B 0,C 180,E1 -10939.956,E2 -10939.956} C_VEL
LIN {X 0,Y 404.143,Z 534.144,A -85,B 0,C 180,E1 -10943.125,E2 -10943.125} C_VEL
LIN {X 0,Y 404.149,Z 534.144,A -85,B 0,C 180,E1 -10946.188,E2 -10946.188} C_VEL
LIN {X 0,Y 404.193,Z 534.284,A -85,B 0,C 180,E1 -10949.538,E2 -10949.538} C_VEL
LIN {X 0,Y 407.147,Z 544.552,A -85,B 0,C 180,E1 -10951.684,E2 -10951.684} C_VEL
LIN {X 0,Y 409.046,Z 553.888,A -85,B 0,C 180,E1 -10953.467,E2 -10953.467} C_VEL
LIN {X 0,Y 408.843,Z 561.864,A -85,B 0,C 180,E1 -10954.821,E2 -10954.821} C_VEL
LIN {X 0,Y 407.649,Z 583.606,A -85,B 0,C 180,E1 -10958.436,E2 -10958.436} C_VEL
LIN {X 0,Y 406.465,Z 606.306,A -85,B 0,C 180,E1 -10962.208,E2 -10962.208} C_VEL
LIN {X 0,Y 406.024,Z 616.928,A -85,B 0,C 180,E1 -10963.954,E2 -10963.954} C_VEL
LIN {X 0,Y 408.164,Z 631.312,A -85,B 0,C 180,E1 -10964.463,E2 -10964.463} C_VEL
LIN {X 0,Y 408.452,Z 637.169,A -85,B 0,C 180,E1 -10964.627,E2 -10964.627} C_VEL
LIN {X 0,Y 407.123,Z 698.265,A -85,B 0,C 180,E1 -10966.046,E2 -10966.046} C_VEL
LIN {X 0,Y 406.734,Z 707.434,A -85,B 0,C 180,E1 -10966.383,E2 -10966.383} C_VEL
